LIN {X 0,Y 573.798,Z 251.946,A -85,B 0,C 180,E1 -2291.656,E2 -2291.656} C_VEL
LIN {X 0,Y 573.261,Z 248.706,A -85,B 0,C 180,E1 -2293.069,E2 -2293.069} C_VEL
LIN {X 0,Y 573.229,Z 248.708,A -85,B 0,C 180,E1 -2295.666,E2 -2295.666} C_VEL
LIN {X 0,Y 573.233,Z 248.709,A -85,B 0,C 180,E1 -2298.543,E2 -2298.543} C_VEL
LIN {X 0,Y 573.247,Z 248.707,A -85,B 0,C 180,E1 -2301.298,E2 -2301.298} C_VEL
LIN {X 0,Y 573.218,Z 248.709,A -85,B 0,C 180,E1 -2304.018,E2 -2304.018} C_VEL
LIN {X 0,Y 573.244,Z 248.707,A -85,B 0,C 180,E1 -2306.516,E2 -2306.516} C_VEL
LIN {X 0,Y 573.235,Z 248.708,A -85,B 0,C 180,E1 -2309.118,E2 -2309.118} C_VEL
LIN {X 0,Y 573.255,Z 248.707,A -85,B 0,C 180,E1 -2311.971,E2 -2311.971} C_VEL
LIN {X 0,Y 573.255,Z 248.705,A -85,B 0,C 180,E1 -2314.589,E2 -2314.589} C_VEL
LIN {X 0,Y 573.239,Z 248.706,A -85,B 0,C 180,E1 -2317.662,E2 -2317.662} C_VEL
LIN {X 0,Y 573.285,Z 248.701,A -85,B 0,C 180,E1 -2320.728,E2 -2320.728} C_VEL
LIN {X 0,Y 573.254,Z 248.706,A -85,B 0,C 180,E1 -2323.621,E2 -2323.621} C_VEL
LIN {X 0,Y 573.271,Z 248.703,A -85,B 0,C 180,E1 -2325.806,E2 -2325.806} C_VEL
LIN {X 0,Y 573.268,Z 248.705,A -85,B 0,C 180,E1 -2328.745,E2 -2328.745} C_VEL
LIN {X 0,Y 573.287,Z 248.701,A -85,B 0,C 180,E1 -2331.54,E2 -2331.54} C_VEL
LIN {X 0,Y 573.293,Z 248.7,A -85,B 0,C 180,E1 -2334.371,E2 -2334.371} C_VEL
LIN {X 0,Y 573.314,Z 248.698,A -85,B 0,C 180,E1 -2337.892,E2 -2337.892} C_VEL
LIN {X 0,Y 573.338,Z 248.694,A -85,B 0,C 180,E1 -2340.702,E2 -2340.702} C_VEL
LIN {X 0,Y 573.235,Z 248.708,A -85,B 0,C 180,E1 -2343.514,E2 -2343.514} C_VEL
LIN {X 0,Y 573.29,Z 248.701,A -85,B 0,C 180,E1 -2345.627,E2 -2345.627} C_VEL
LIN {X 0,Y 573.287,Z 248.703,A -85,B 0,C 180,E1 -2348.459,E2 -2348.459} C_VEL
LIN {X 0,Y 573.275,Z 248.702,A -85,B 0,C 180,E1 -2351.311,E2 -2351.311} C_VEL
LIN {X 0,Y 573.284,Z 248.701,A -85,B 0,C 180,E1 -2354.423,E2 -2354.423} C_VEL
LIN {X 0,Y 573.261,Z 248.705,A -85,B 0,C 180,E1 -2357.11,E2 -2357.11} C_VEL
LIN {X 0,Y 573.242,Z 248.709,A -85,B 0,C 180,E1 -2360.076,E2 -2360.076} C_VEL
LIN {X 0,Y 573.237,Z 248.708,A -85,B 0,C 180,E1 -2362.337,E2 -2362.337} C_VEL
LIN {X 0,Y 573.25,Z 248.704,A -85,B 0,C 180,E1 -2364.387,E2 -2364.387} C_VEL
LIN {X 0,Y 572.623,Z 248.784,A -85,B 0,C 180,E1 -2364.973,E2 -2364.973} C_VEL
LIN {X 0,Y 569.781,Z 249.141,A -85,B 0,C 180,E1 -2365.924,E2 -2365.924} C_VEL
LIN {X 0,Y 567.351,Z 249.444,A -85,B 0,C 180,E1 -2366.69,E2 -2366.69} C_VEL
LIN {X 0,Y 566.3,Z 249.573,A -85,B 0,C 180,E1 -2367.281,E2 -2367.281} C_VEL
LIN {X 0,Y 566.212,Z 249.582,A -85,B 0,C 180,E1 -2367.481,E2 -2367.481} C_VEL
LIN {X 0,Y 566.201,Z 249.584,A -85,B 0,C 180,E1 -2369.768,E2 -2369.768} C_VEL
LIN {X 0,Y 566.205,Z 249.584,A -85,B 0,C 180,E1 -2372.429,E2 -2372.429} C_VEL
LIN {X 0,Y 566.212,Z 249.582,A -85,B 0,C 180,E1 -2374.993,E2 -2374.993} C_VEL
LIN {X 0,Y 566.194,Z 249.584,A -85,B 0,C 180,E1 -2377.46,E2 -2377.46} C_VEL
LIN {X 0,Y 566.223,Z 249.581,A -85,B 0,C 180,E1 -2380.196,E2 -2380.196} C_VEL
LIN {X 0,Y 566.201,Z 249.585,A -85,B 0,C 180,E1 -2383.053,E2 -2383.053} C_VEL
LIN {X 0,Y 566.198,Z 249.585,A -85,B 0,C 180,E1 -2386.047,E2 -2386.047} C_VEL
LIN {X 0,Y 566.207,Z 249.582,A -85,B 0,C 180,E1 -2388.863,E2 -2388.863} C_VEL
LIN {X 0,Y 566.184,Z 249.587,A -85,B 0,C 180,E1 -2391.636,E2 -2391.636} C_VEL
LIN {X 0,Y 566.205,Z 249.584,A -85,B 0,C 180,E1 -2394.311,E2 -2394.311} C_VEL
LIN {X 0,Y 566.222,Z 249.581,A -85,B 0,C 180,E1 -2396.898,E2 -2396.898} C_VEL
LIN {X 0,Y 566.188,Z 249.585,A -85,B 0,C 180,E1 -2399.407,E2 -2399.407} C_VEL
LIN {X 0,Y 566.22,Z 249.584,A -85,B 0,C 180,E1 -2401.857,E2 -2401.857} C_VEL
LIN {X 0,Y 566.217,Z 249.581,A -85,B 0,C 180,E1 -2404.251,E2 -2404.251} C_VEL
LIN {X 0,Y 566.184,Z 249.585,A -85,B 0,C 180,E1 -2406.712,E2 -2406.712} C_VEL
LIN {X 0,Y 566.211,Z 249.582,A -85,B 0,C 180,E1 -2409.662,E2 -2409.662} C_VEL
LIN {X 0,Y 566.195,Z 249.584,A -85,B 0,C 180,E1 -2412.668,E2 -2412.668} C_VEL
LIN {X 0,Y 566.224,Z 249.582,A -85,B 0,C 180,E1 -2415.626,E2 -2415.626} C_VEL
LIN {X 0,Y 566.265,Z 249.577,A -85,B 0,C 180,E1 -2418.653,E2 -2418.653} C_VEL
LIN {X 0,Y 566.241,Z 249.579,A -85,B 0,C 180,E1 -2421.434,E2 -2421.434} C_VEL
LIN {X 0,Y 566.254,Z 249.576,A -85,B 0,C 180,E1 -2424.301,E2 -2424.301} C_VEL
LIN {X 0,Y 566.012,Z 249.791,A -85,B 0,C 180,E1 -2426.44,E2 -2426.44} C_VEL
LIN {X 0,Y 566.132,Z 252.646,A -85,B 0,C 180,E1 -2429.288,E2 -2429.288} C_VEL
LIN {X 0,Y 566.053,Z 254.767,A -85,B 0,C 180,E1 -2431.422,E2 -2431.422} C_VEL
LIN {X 0,Y 565.952,Z 257.617,A -85,B 0,C 180,E1 -2434.272,E2 -2434.272} C_VEL
LIN {X 0,Y 565.964,Z 260.459,A -85,B 0,C 180,E1 -2437.133,E2 -2437.133} C_VEL
LIN {X 0,Y 565.884,Z 263.341,A -85,B 0,C 180,E1 -2440.013,E2 -2440.013} C_VEL
LIN {X 0,Y 565.869,Z 265.835,A -85,B 0,C 180,E1 -2442.188,E2 -2442.188} C_VEL
LIN {X 0,Y 565.846,Z 269.385,A -85,B 0,C 180,E1 -2445.234,E2 -2445.234} C_VEL
LIN {X 0,Y 567.922,Z 278.23,A -85,B 0,C 180,E1 -2445.452,E2 -2445.452} C_VEL
LIN {X 0,Y 567.738,Z 293.829,A -85,B 0,C 180,E1 -2445.826,E2 -2445.826} C_VEL
LIN {X 0,Y 567.531,Z 308.287,A -85,B 0,C 180,E1 -2446.316,E2 -2446.316} C_VEL
LIN {X 0,Y 567.321,Z 322.051,A -85,B 0,C 180,E1 -2446.924,E2 -2446.924} C_VEL
LIN {X 0,Y 567.111,Z 335.614,A -85,B 0,C 180,E1 -2447.674,E2 -2447.674} C_VEL
LIN {X 0,Y 566.885,Z 349.436,A -85,B 0,C 180,E1 -2448.616,E2 -2448.616} C_VEL
LIN {X 0,Y 566.624,Z 362.05,A -85,B 0,C 180,E1 -2449.659,E2 -2449.659} C_VEL
LIN {X 0,Y 566.445,Z 372.696,A -85,B 0,C 180,E1 -2450.707,E2 -2450.707} C_VEL
LIN {X 0,Y 566.258,Z 382.584,A -85,B 0,C 180,E1 -2451.859,E2 -2451.859} C_VEL
LIN {X 0,Y 566.15,Z 391.619,A -85,B 0,C 180,E1 -2453.115,E2 -2453.115} C_VEL
LIN {X 0,Y 566.024,Z 400.309,A -85,B 0,C 180,E1 -2454.579,E2 -2454.579} C_VEL
LIN {X 0,Y 565.983,Z 406.016,A -85,B 0,C 180,E1 -2455.76,E2 -2455.76} C_VEL
LIN {X 0,Y 565.926,Z 410.812,A -85,B 0,C 180,E1 -2456.953,E2 -2456.953} C_VEL
LIN {X 0,Y 565.893,Z 415.77,A -85,B 0,C 180,E1 -2458.564,E2 -2458.564} C_VEL
LIN {X 0,Y 565.857,Z 418.497,A -85,B 0,C 180,E1 -2459.788,E2 -2459.788} C_VEL
LIN {X 0,Y 565.854,Z 420.317,A -85,B 0,C 180,E1 -2461.022,E2 -2461.022} C_VEL
LIN {X 0,Y 565.833,Z 421.357,A -85,B 0,C 180,E1 -2462.373,E2 -2462.373} C_VEL
LIN {X 0,Y 565.854,Z 421.235,A -85,B 0,C 180,E1 -2463.98,E2 -2463.98} C_VEL
LIN {X 0,Y 565.843,Z 420.456,A -85,B 0,C 180,E1 -2464.943,E2 -2464.943} C_VEL
LIN {X 0,Y 565.855,Z 417.91,A -85,B 0,C 180,E1 -2466.595,E2 -2466.595} C_VEL
LIN {X 0,Y 565.9,Z 414.68,A -85,B 0,C 180,E1 -2467.933,E2 -2467.933} C_VEL
LIN {X 0,Y 565.934,Z 410.254,A -85,B 0,C 180,E1 -2469.296,E2 -2469.296} C_VEL
LIN {X 0,Y 565.965,Z 404.088,A -85,B 0,C 180,E1 -2470.759,E2 -2470.759} C_VEL
LIN {X 0,Y 566.033,Z 397.007,A -85,B 0,C 180,E1 -2472.103,E2 -2472.103} C_VEL
LIN {X 0,Y 566.146,Z 389.512,A -85,B 0,C 180,E1 -2473.285,E2 -2473.285} C_VEL
LIN {X 0,Y 566.314,Z 380.208,A -85,B 0,C 180,E1 -2474.52,E2 -2474.52} C_VEL
LIN {X 0,Y 566.505,Z 369.066,A -85,B 0,C 180,E1 -2475.756,E2 -2475.756} C_VEL
LIN {X 0,Y 566.73,Z 358.35,A -85,B 0,C 180,E1 -2476.754,E2 -2476.754} C_VEL
LIN {X 0,Y 566.928,Z 345.77,A -85,B 0,C 180,E1 -2477.74,E2 -2477.74} C_VEL
LIN {X 0,Y 567.174,Z 332.538,A -85,B 0,C 180,E1 -2478.596,E2 -2478.596} C_VEL
LIN {X 0,Y 567.408,Z 318.734,A -85,B 0,C 180,E1 -2479.323,E2 -2479.323} C_VEL
LIN {X 0,Y 567.632,Z 304.228,A -85,B 0,C 180,E1 -2479.924,E2 -2479.924} C_VEL
LIN {X 0,Y 567.847,Z 289.312,A -85,B 0,C 180,E1 -2480.387,E2 -2480.387} C_VEL
LIN {X 0,Y 567.764,Z 277.487,A -85,B 0,C 180,E1 -2480.658,E2 -2480.658} C_VEL
LIN {X 0,Y 565.864,Z 269.366,A -85,B 0,C 180,E1 -2480.872,E2 -2480.872} C_VEL
LIN {X 0,Y 565.876,Z 265.917,A -85,B 0,C 180,E1 -2483.83,E2 -2483.83} C_VEL
LIN {X 0,Y 565.881,Z 262.494,A -85,B 0,C 180,E1 -2486.877,E2 -2486.877} C_VEL
LIN {X 0,Y 565.941,Z 260.154,A -85,B 0,C 180,E1 -2489.394,E2 -2489.394} C_VEL
LIN {X 0,Y 565.985,Z 257.918,A -85,B 0,C 180,E1 -2491.846,E2 -2491.846} C_VEL
LIN {X 0,Y 566.067,Z 254.853,A -85,B 0,C 180,E1 -2495.032,E2 -2495.032} C_VEL
LIN {X 0,Y 566.028,Z 252.512,A -85,B 0,C 180,E1 -2497.363,E2 -2497.363} C_VEL
LIN {X 0,Y 566.053,Z 250.266,A -85,B 0,C 180,E1 -2499.658,E2 -2499.658} C_VEL
LIN {X 0,Y 566.089,Z 249.601,A -85,B 0,C 180,E1 -2500.653,E2 -2500.653} C_VEL
LIN {X 0,Y 566.215,Z 249.585,A -85,B 0,C 180,E1 -2503.413,E2 -2503.413} C_VEL
LIN {X 0,Y 566.194,Z 249.585,A -85,B 0,C 180,E1 -2506.36,E2 -2506.36} C_VEL
LIN {X 0,Y 566.228,Z 249.582,A -85,B 0,C 180,E1 -2508.676,E2 -2508.676} C_VEL
LIN {X 0,Y 566.231,Z 249.58,A -85,B 0,C 180,E1 -2511.435,E2 -2511.435} C_VEL
LIN {X 0,Y 566.257,Z 249.577,A -85,B 0,C 180,E1 -2514.303,E2 -2514.303} C_VEL
LIN {X 0,Y 566.28,Z 249.573,A -85,B 0,C 180,E1 -2517.867,E2 -2517.867} C_VEL
LIN {X 0,Y 566.3,Z 249.571,A -85,B 0,C 180,E1 -2520.712,E2 -2520.712} C_VEL
LIN {X 0,Y 566.273,Z 249.575,A -85,B 0,C 180,E1 -2522.846,E2 -2522.846} C_VEL
LIN {X 0,Y 566.258,Z 249.578,A -85,B 0,C 180,E1 -2525.699,E2 -2525.699} C_VEL
LIN {X 0,Y 566.232,Z 249.58,A -85,B 0,C 180,E1 -2528.566,E2 -2528.566} C_VEL
LIN {X 0,Y 566.239,Z 249.578,A -85,B 0,C 180,E1 -2531.455,E2 -2531.455} C_VEL
LIN {X 0,Y 566.232,Z 249.579,A -85,B 0,C 180,E1 -2534.508,E2 -2534.508} C_VEL
LIN {X 0,Y 566.197,Z 249.586,A -85,B 0,C 180,E1 -2537.332,E2 -2537.332} C_VEL
LIN {X 0,Y 566.217,Z 249.583,A -85,B 0,C 180,E1 -2540.338,E2 -2540.338} C_VEL
LIN {X 0,Y 566.187,Z 249.586,A -85,B 0,C 180,E1 -2543.404,E2 -2543.404} C_VEL
LIN {X 0,Y 566.225,Z 249.583,A -85,B 0,C 180,E1 -2545.749,E2 -2545.749} C_VEL
LIN {X 0,Y 566.2,Z 249.584,A -85,B 0,C 180,E1 -2548.203,E2 -2548.203} C_VEL
LIN {X 0,Y 566.189,Z 249.588,A -85,B 0,C 180,E1 -2551.077,E2 -2551.077} C_VEL
LIN {X 0,Y 566.21,Z 249.584,A -85,B 0,C 180,E1 -2553.735,E2 -2553.735} C_VEL
LIN {X 0,Y 566.198,Z 249.586,A -85,B 0,C 180,E1 -2556.57,E2 -2556.57} C_VEL
LIN {X 0,Y 566.22,Z 249.584,A -85,B 0,C 180,E1 -2559.274,E2 -2559.274} C_VEL
LIN {X 0,Y 566.188,Z 249.586,A -85,B 0,C 180,E1 -2562.09,E2 -2562.09} C_VEL
LIN {X 0,Y 566.172,Z 249.588,A -85,B 0,C 180,E1 -2565.036,E2 -2565.036} C_VEL
LIN {X 0,Y 566.255,Z 249.786,A -85,B 0,C 180,E1 -2566.83,E2 -2566.83} C_VEL
LIN {X 0,Y 566.928,Z 254.966,A -85,B 0,C 180,E1 -2568.928,E2 -2568.928} C_VEL
LIN {X 0,Y 566.868,Z 262.764,A -85,B 0,C 180,E1 -2571.692,E2 -2571.692} C_VEL
LIN {X 0,Y 566.755,Z 270.211,A -85,B 0,C 180,E1 -2574.352,E2 -2574.352} C_VEL
LIN {X 0,Y 566.609,Z 277.638,A -85,B 0,C 180,E1 -2576.924,E2 -2576.924} C_VEL
LIN {X 0,Y 566.513,Z 286.302,A -85,B 0,C 180,E1 -2579.84,E2 -2579.84} C_VEL
LIN {X 0,Y 566.398,Z 294.967,A -85,B 0,C 180,E1 -2582.671,E2 -2582.671} C_VEL
LIN {X 0,Y 566.297,Z 303.632,A -85,B 0,C 180,E1 -2585.434,E2 -2585.434} C_VEL
LIN {X 0,Y 566.232,Z 312.296,A -85,B 0,C 180,E1 -2588.14,E2 -2588.14} C_VEL
LIN {X 0,Y 566.146,Z 320.449,A -85,B 0,C 180,E1 -2590.639,E2 -2590.639} C_VEL
LIN {X 0,Y 566.121,Z 325.422,A -85,B 0,C 180,E1 -2592.146,E2 -2592.146} C_VEL
LIN {X 0,Y 567.997,Z 334.459,A -85,B 0,C 180,E1 -2592.341,E2 -2592.341} C_VEL
LIN {X 0,Y 567.864,Z 349.029,A -85,B 0,C 180,E1 -2592.652,E2 -2592.652} C_VEL
LIN {X 0,Y 567.703,Z 363.222,A -85,B 0,C 180,E1 -2593.087,E2 -2593.087} C_VEL
LIN {X 0,Y 567.453,Z 376.838,A -85,B 0,C 180,E1 -2593.635,E2 -2593.635} C_VEL
LIN {X 0,Y 567.219,Z 391.115,A -85,B 0,C 180,E1 -2594.367,E2 -2594.367} C_VEL
LIN {X 0,Y 566.95,Z 404.54,A -85,B 0,C 180,E1 -2595.217,E2 -2595.217} C_VEL
LIN {X 0,Y 566.756,Z 417.173,A -85,B 0,C 180,E1 -2596.19,E2 -2596.19} C_VEL
LIN {X 0,Y 566.545,Z 428.978,A -85,B 0,C 180,E1 -2597.28,E2 -2597.28} C_VEL
LIN {X 0,Y 566.343,Z 438.905,A -85,B 0,C 180,E1 -2598.367,E2 -2598.367} C_VEL
LIN {X 0,Y 566.204,Z 448.622,A -85,B 0,C 180,E1 -2599.632,E2 -2599.632} C_VEL
LIN {X 0,Y 566.079,Z 456.723,A -85,B 0,C 180,E1 -2600.893,E2 -2600.893} C_VEL
LIN {X 0,Y 566.014,Z 463.428,A -85,B 0,C 180,E1 -2602.15,E2 -2602.15} C_VEL
LIN {X 0,Y 565.943,Z 469.609,A -85,B 0,C 180,E1 -2603.584,E2 -2603.584} C_VEL
LIN {X 0,Y 565.867,Z 474.386,A -85,B 0,C 180,E1 -2605.013,E2 -2605.013} C_VEL
LIN {X 0,Y 565.91,Z 477.889,A -85,B 0,C 180,E1 -2606.44,E2 -2606.44} C_VEL
LIN {X 0,Y 565.839,Z 480.194,A -85,B 0,C 180,E1 -2607.865,E2 -2607.865} C_VEL
LIN {X 0,Y 565.837,Z 481.35,A -85,B 0,C 180,E1 -2609.289,E2 -2609.289} C_VEL
LIN {X 0,Y 565.837,Z 481.349,A -85,B 0,C 180,E1 -2610.712,E2 -2610.712} C_VEL
LIN {X 0,Y 565.839,Z 480.192,A -85,B 0,C 180,E1 -2612.136,E2 -2612.136} C_VEL
LIN {X 0,Y 565.91,Z 477.885,A -85,B 0,C 180,E1 -2613.561,E2 -2613.561} C_VEL
LIN {X 0,Y 565.867,Z 474.383,A -85,B 0,C 180,E1 -2614.988,E2 -2614.988} C_VEL
LIN {X 0,Y 565.959,Z 470.923,A -85,B 0,C 180,E1 -2616.059,E2 -2616.059} C_VEL
LIN {X 0,Y 565.998,Z 465.085,A -85,B 0,C 180,E1 -2617.492,E2 -2617.492} C_VEL
LIN {X 0,Y 566.057,Z 457.727,A -85,B 0,C 180,E1 -2618.929,E2 -2618.929} C_VEL
LIN {X 0,Y 566.209,Z 449.853,A -85,B 0,C 180,E1 -2620.188,E2 -2620.188} C_VEL
LIN {X 0,Y 566.31,Z 440.386,A -85,B 0,C 180,E1 -2621.453,E2 -2621.453} C_VEL
LIN {X 0,Y 566.492,Z 430.744,A -85,B 0,C 180,E1 -2622.54,E2 -2622.54} C_VEL
LIN {X 0,Y 566.671,Z 419.283,A -85,B 0,C 180,E1 -2623.63,E2 -2623.63} C_VEL
LIN {X 0,Y 566.929,Z 406.663,A -85,B 0,C 180,E1 -2624.631,E2 -2624.631} C_VEL
LIN {X 0,Y 567.147,Z 394.229,A -85,B 0,C 180,E1 -2625.452,E2 -2625.452} C_VEL
LIN {X 0,Y 567.382,Z 380.751,A -85,B 0,C 180,E1 -2626.183,E2 -2626.183} C_VEL
LIN {X 0,Y 567.634,Z 367.038,A -85,B 0,C 180,E1 -2626.777,E2 -2626.777} C_VEL
LIN {X 0,Y 567.84,Z 351.699,A -85,B 0,C 180,E1 -2627.28,E2 -2627.28} C_VEL
LIN {X 0,Y 567.962,Z 336.542,A -85,B 0,C 180,E1 -2627.626,E2 -2627.626} C_VEL
LIN {X 0,Y 567.707,Z 332.422,A -85,B 0,C 180,E1 -2627.7,E2 -2627.7} C_VEL
LIN {X 0,Y 566.119,Z 325.381,A -85,B 0,C 180,E1 -2627.867,E2 -2627.867} C_VEL
LIN {X 0,Y 566.177,Z 316.006,A -85,B 0,C 180,E1 -2630.719,E2 -2630.719} C_VEL
LIN {X 0,Y 566.31,Z 306.104,A -85,B 0,C 180,E1 -2633.787,E2 -2633.787} C_VEL
LIN {X 0,Y 566.381,Z 296.939,A -85,B 0,C 180,E1 -2636.694,E2 -2636.694} C_VEL
LIN {X 0,Y 566.492,Z 288.814,A -85,B 0,C 180,E1 -2639.331,E2 -2639.331} C_VEL
LIN {X 0,Y 566.566,Z 280.11,A -85,B 0,C 180,E1 -2642.236,E2 -2642.236} C_VEL
LIN {X 0,Y 566.683,Z 271.893,A -85,B 0,C 180,E1 -2645.062,E2 -2645.062} C_VEL
LIN {X 0,Y 566.89,Z 263.99,A -85,B 0,C 180,E1 -2647.856,E2 -2647.856} C_VEL
LIN {X 0,Y 566.923,Z 257.616,A -85,B 0,C 180,E1 -2650.138,E2 -2650.138} C_VEL
LIN {X 0,Y 566.759,Z 252.805,A -85,B 0,C 180,E1 -2651.925,E2 -2651.925} C_VEL
LIN {X 0,Y 566.225,Z 249.583,A -85,B 0,C 180,E1 -2653.296,E2 -2653.296} C_VEL
LIN {X 0,Y 566.199,Z 249.584,A -85,B 0,C 180,E1 -2656.049,E2 -2656.049} C_VEL
LIN {X 0,Y 566.208,Z 249.584,A -85,B 0,C 180,E1 -2659.215,E2 -2659.215} C_VEL
LIN {X 0,Y 566.19,Z 249.586,A -85,B 0,C 180,E1 -2661.637,E2 -2661.637} C_VEL
LIN {X 0,Y 566.168,Z 249.588,A -85,B 0,C 180,E1 -2664.308,E2 -2664.308} C_VEL
LIN {X 0,Y 566.209,Z 249.584,A -85,B 0,C 180,E1 -2666.897,E2 -2666.897} C_VEL
LIN {X 0,Y 566.186,Z 249.585,A -85,B 0,C 180,E1 -2669.407,E2 -2669.407} C_VEL
LIN {X 0,Y 566.217,Z 249.583,A -85,B 0,C 180,E1 -2671.857,E2 -2671.857} C_VEL
LIN {X 0,Y 566.215,Z 249.583,A -85,B 0,C 180,E1 -2674.251,E2 -2674.251} C_VEL
LIN {X 0,Y 566.178,Z 249.586,A -85,B 0,C 180,E1 -2676.718,E2 -2676.718} C_VEL
LIN {X 0,Y 566.218,Z 249.581,A -85,B 0,C 180,E1 -2679.662,E2 -2679.662} C_VEL
LIN {X 0,Y 566.205,Z 249.584,A -85,B 0,C 180,E1 -2682.668,E2 -2682.668} C_VEL
LIN {X 0,Y 566.234,Z 249.581,A -85,B 0,C 180,E1 -2685.626,E2 -2685.626} C_VEL
LIN {X 0,Y 566.24,Z 249.581,A -85,B 0,C 180,E1 -2688.675,E2 -2688.675} C_VEL
LIN {X 0,Y 566.231,Z 249.579,A -85,B 0,C 180,E1 -2691.434,E2 -2691.434} C_VEL
LIN {X 0,Y 566.26,Z 249.576,A -85,B 0,C 180,E1 -2694.301,E2 -2694.301} C_VEL
LIN {X 0,Y 566.285,Z 249.573,A -85,B 0,C 180,E1 -2697.866,E2 -2697.866} C_VEL
LIN {X 0,Y 566.308,Z 249.57,A -85,B 0,C 180,E1 -2700.71,E2 -2700.71} C_VEL
LIN {X 0,Y 566.276,Z 249.574,A -85,B 0,C 180,E1 -2702.845,E2 -2702.845} C_VEL
LIN {X 0,Y 566.259,Z 249.577,A -85,B 0,C 180,E1 -2705.697,E2 -2705.697} C_VEL
LIN {X 0,Y 566.23,Z 249.582,A -85,B 0,C 180,E1 -2708.565,E2 -2708.565} C_VEL
LIN {X 0,Y 566.245,Z 249.578,A -85,B 0,C 180,E1 -2711.453,E2 -2711.453} C_VEL
LIN {X 0,Y 566.237,Z 249.58,A -85,B 0,C 180,E1 -2714.506,E2 -2714.506} C_VEL
LIN {X 0,Y 566.205,Z 249.583,A -85,B 0,C 180,E1 -2717.33,E2 -2717.33} C_VEL
LIN {X 0,Y 566.208,Z 249.583,A -85,B 0,C 180,E1 -2720.336,E2 -2720.336} C_VEL
LIN {X 0,Y 566.19,Z 249.586,A -85,B 0,C 180,E1 -2723.403,E2 -2723.403} C_VEL
LIN {X 0,Y 566.214,Z 249.582,A -85,B 0,C 180,E1 -2725.748,E2 -2725.748} C_VEL
LIN {X 0,Y 566.212,Z 249.582,A -85,B 0,C 180,E1 -2727.481,E2 -2727.481} C_VEL
LIN {X 0,Y 565.535,Z 249.668,A -85,B 0,C 180,E1 -2728.075,E2 -2728.075} C_VEL
LIN {X 0,Y 562.666,Z 250.023,A -85,B 0,C 180,E1 -2729.038,E2 -2729.038} C_VEL
LIN {X 0,Y 560.251,Z 250.325,A -85,B 0,C 180,E1 -2729.814,E2 -2729.814} C_VEL
LIN {X 0,Y 559.221,Z 250.455,A -85,B 0,C 180,E1 -2730.413,E2 -2730.413} C_VEL
LIN {X 0,Y 559.141,Z 250.461,A -85,B 0,C 180,E1 -2730.615,E2 -2730.615} C_VEL
LIN {X 0,Y 559.163,Z 250.461,A -85,B 0,C 180,E1 -2733.573,E2 -2733.573} C_VEL
LIN {X 0,Y 559.167,Z 250.46,A -85,B 0,C 180,E1 -2736.447,E2 -2736.447} C_VEL
LIN {X 0,Y 559.175,Z 250.46,A -85,B 0,C 180,E1 -2738.932,E2 -2738.932} C_VEL
LIN {X 0,Y 559.188,Z 250.458,A -85,B 0,C 180,E1 -2741.766,E2 -2741.766} C_VEL
LIN {X 0,Y 559.135,Z 250.463,A -85,B 0,C 180,E1 -2744.738,E2 -2744.738} C_VEL
LIN {X 0,Y 559.162,Z 250.462,A -85,B 0,C 180,E1 -2747.256,E2 -2747.256} C_VEL
LIN {X 0,Y 559.181,Z 250.459,A -85,B 0,C 180,E1 -2750.134,E2 -2750.134} C_VEL
LIN {X 0,Y 559.14,Z 250.462,A -85,B 0,C 180,E1 -2752.891,E2 -2752.891} C_VEL
LIN {X 0,Y 559.149,Z 250.464,A -85,B 0,C 180,E1 -2755.555,E2 -2755.555} C_VEL
LIN {X 0,Y 559.166,Z 250.46,A -85,B 0,C 180,E1 -2758.137,E2 -2758.137} C_VEL
LIN {X 0,Y 559.151,Z 250.462,A -85,B 0,C 180,E1 -2760.646,E2 -2760.646} C_VEL
LIN {X 0,Y 559.175,Z 250.459,A -85,B 0,C 180,E1 -2763.169,E2 -2763.169} C_VEL
LIN {X 0,Y 559.149,Z 250.462,A -85,B 0,C 180,E1 -2765.494,E2 -2765.494} C_VEL
LIN {X 0,Y 559.168,Z 250.459,A -85,B 0,C 180,E1 -2768.623,E2 -2768.623} C_VEL
LIN {X 0,Y 559.163,Z 250.46,A -85,B 0,C 180,E1 -2770.926,E2 -2770.926} C_VEL
LIN {X 0,Y 559.162,Z 250.46,A -85,B 0,C 180,E1 -2773.947,E2 -2773.947} C_VEL
LIN {X 0,Y 559.166,Z 250.46,A -85,B 0,C 180,E1 -2776.183,E2 -2776.183} C_VEL
LIN {X 0,Y 559.202,Z 250.455,A -85,B 0,C 180,E1 -2779.133,E2 -2779.133} C_VEL
LIN {X 0,Y 559.204,Z 250.454,A -85,B 0,C 180,E1 -2782.053,E2 -2782.053} C_VEL
LIN {X 0,Y 559.214,Z 250.456,A -85,B 0,C 180,E1 -2784.952,E2 -2784.952} C_VEL
LIN {X 0,Y 558.951,Z 250.49,A -85,B 0,C 180,E1 -2786.395,E2 -2786.395} C_VEL
LIN {X 0,Y 559.086,Z 253.286,A -85,B 0,C 180,E1 -2789.279,E2 -2789.279} C_VEL
LIN {X 0,Y 558.997,Z 255.438,A -85,B 0,C 180,E1 -2791.44,E2 -2791.44} C_VEL
LIN {X 0,Y 558.884,Z 258.3,A -85,B 0,C 180,E1 -2794.327,E2 -2794.327} C_VEL
LIN {X 0,Y 558.875,Z 261.141,A -85,B 0,C 180,E1 -2797.224,E2 -2797.224} C_VEL
LIN {X 0,Y 558.817,Z 263.981,A -85,B 0,C 180,E1 -2800.141,E2 -2800.141} C_VEL
LIN {X 0,Y 558.771,Z 266.33,A -85,B 0,C 180,E1 -2802.346,E2 -2802.346} C_VEL
LIN {X 0,Y 558.743,Z 269.365,A -85,B 0,C 180,E1 -2804.982,E2 -2804.982} C_VEL
LIN {X 0,Y 561.182,Z 279.993,A -85,B 0,C 180,E1 -2805.27,E2 -2805.27} C_VEL
LIN {X 0,Y 560.937,Z 295.094,A -85,B 0,C 180,E1 -2805.649,E2 -2805.649} C_VEL
LIN {X 0,Y 560.679,Z 310.405,A -85,B 0,C 180,E1 -2806.194,E2 -2806.194} C_VEL
LIN {X 0,Y 560.416,Z 324.608,A -85,B 0,C 180,E1 -2806.856,E2 -2806.856} C_VEL
LIN {X 0,Y 560.162,Z 338.641,A -85,B 0,C 180,E1 -2807.677,E2 -2807.677} C_VEL
LIN {X 0,Y 559.929,Z 351.182,A -85,B 0,C 180,E1 -2808.571,E2 -2808.571} C_VEL
LIN {X 0,Y 559.608,Z 363.537,A -85,B 0,C 180,E1 -2809.63,E2 -2809.63} C_VEL
LIN {X 0,Y 559.426,Z 374.786,A -85,B 0,C 180,E1 -2810.787,E2 -2810.787} C_VEL
LIN {X 0,Y 559.227,Z 384.6,A -85,B 0,C 180,E1 -2811.987,E2 -2811.987} C_VEL
LIN {X 0,Y 559.101,Z 392.793,A -85,B 0,C 180,E1 -2813.174,E2 -2813.174} C_VEL
LIN {X 0,Y 558.949,Z 400.53,A -85,B 0,C 180,E1 -2814.514,E2 -2814.514} C_VEL
LIN {X 0,Y 558.908,Z 406.206,A -85,B 0,C 180,E1 -2815.71,E2 -2815.71} C_VEL
LIN {X 0,Y 558.836,Z 410.961,A -85,B 0,C 180,E1 -2816.919,E2 -2816.919} C_VEL
LIN {X 0,Y 558.795,Z 415.876,A -85,B 0,C 180,E1 -2818.55,E2 -2818.55} C_VEL
LIN {X 0,Y 558.77,Z 419.252,A -85,B 0,C 180,E1 -2820.205,E2 -2820.205} C_VEL
LIN {X 0,Y 558.75,Z 420.548,A -85,B 0,C 180,E1 -2821.209,E2 -2821.209} C_VEL
LIN {X 0,Y 558.745,Z 421.441,A -85,B 0,C 180,E1 -2822.742,E2 -2822.742} C_VEL
LIN {X 0,Y 558.76,Z 421.301,A -85,B 0,C 180,E1 -2823.89,E2 -2823.89} C_VEL
LIN {X 0,Y 558.74,Z 420.032,A -85,B 0,C 180,E1 -2825.352,E2 -2825.352} C_VEL
LIN {X 0,Y 558.749,Z 418.404,A -85,B 0,C 180,E1 -2826.392,E2 -2826.392} C_VEL
LIN {X 0,Y 558.776,Z 415.746,A -85,B 0,C 180,E1 -2827.594,E2 -2827.594} C_VEL
LIN {X 0,Y 558.851,Z 411.68,A -85,B 0,C 180,E1 -2828.96,E2 -2828.96} C_VEL
LIN {X 0,Y 558.894,Z 406.298,A -85,B 0,C 180,E1 -2830.36,E2 -2830.36} C_VEL
LIN {X 0,Y 558.947,Z 399.385,A -85,B 0,C 180,E1 -2831.789,E2 -2831.789} C_VEL
LIN {X 0,Y 559.102,Z 391.002,A -85,B 0,C 180,E1 -2833.193,E2 -2833.193} C_VEL
LIN {X 0,Y 559.262,Z 381.909,A -85,B 0,C 180,E1 -2834.456,E2 -2834.456} C_VEL
LIN {X 0,Y 559.445,Z 372.126,A -85,B 0,C 180,E1 -2835.602,E2 -2835.602} C_VEL
LIN {X 0,Y 559.712,Z 360.509,A -85,B 0,C 180,E1 -2836.741,E2 -2836.741} C_VEL
LIN {X 0,Y 559.992,Z 347.925,A -85,B 0,C 180,E1 -2837.77,E2 -2837.77} C_VEL
LIN {X 0,Y 560.271,Z 335.564,A -85,B 0,C 180,E1 -2838.611,E2 -2838.611} C_VEL
LIN {X 0,Y 560.537,Z 321.602,A -85,B 0,C 180,E1 -2839.39,E2 -2839.39} C_VEL
LIN {X 0,Y 560.778,Z 306.826,A -85,B 0,C 180,E1 -2840.041,E2 -2840.041} C_VEL
LIN {X 0,Y 561.029,Z 291.201,A -85,B 0,C 180,E1 -2840.555,E2 -2840.555} C_VEL
LIN {X 0,Y 561.046,Z 278.888,A -85,B 0,C 180,E1 -2840.847,E2 -2840.847} C_VEL
LIN {X 0,Y 558.796,Z 269.372,A -85,B 0,C 180,E1 -2841.1,E2 -2841.1} C_VEL
LIN {X 0,Y 558.802,Z 266.305,A -85,B 0,C 180,E1 -2843.765,E2 -2843.765} C_VEL
LIN {X 0,Y 558.831,Z 263.59,A -85,B 0,C 180,E1 -2846.404,E2 -2846.404} C_VEL
LIN {X 0,Y 558.88,Z 261.221,A -85,B 0,C 180,E1 -2848.965,E2 -2848.965} C_VEL
LIN {X 0,Y 558.928,Z 258.728,A -85,B 0,C 180,E1 -2851.663,E2 -2851.663} C_VEL
LIN {X 0,Y 558.982,Z 255.666,A -85,B 0,C 180,E1 -2854.855,E2 -2854.855} C_VEL
LIN {X 0,Y 558.995,Z 253.566,A -85,B 0,C 180,E1 -2857.062,E2 -2857.062} C_VEL
LIN {X 0,Y 558.983,Z 251.27,A -85,B 0,C 180,E1 -2859.389,E2 -2859.389} C_VEL
LIN {X 0,Y 559,Z 250.536,A -85,B 0,C 180,E1 -2860.157,E2 -2860.157} C_VEL
LIN {X 0,Y 559.164,Z 250.461,A -85,B 0,C 180,E1 -2862.787,E2 -2862.787} C_VEL
LIN {X 0,Y 559.189,Z 250.459,A -85,B 0,C 180,E1 -2865.443,E2 -2865.443} C_VEL
LIN {X 0,Y 559.199,Z 250.457,A -85,B 0,C 180,E1 -2868.605,E2 -2868.605} C_VEL
LIN {X 0,Y 559.189,Z 250.457,A -85,B 0,C 180,E1 -2871.327,E2 -2871.327} C_VEL
LIN {X 0,Y 559.227,Z 250.453,A -85,B 0,C 180,E1 -2874.231,E2 -2874.231} C_VEL
LIN {X 0,Y 559.251,Z 250.449,A -85,B 0,C 180,E1 -2877.84,E2 -2877.84} C_VEL
LIN {X 0,Y 559.27,Z 250.447,A -85,B 0,C 180,E1 -2880.721,E2 -2880.721} C_VEL
LIN {X 0,Y 559.239,Z 250.451,A -85,B 0,C 180,E1 -2882.882,E2 -2882.882} C_VEL
LIN {X 0,Y 559.227,Z 250.453,A -85,B 0,C 180,E1 -2885.771,E2 -2885.771} C_VEL
LIN {X 0,Y 559.19,Z 250.458,A -85,B 0,C 180,E1 -2888.675,E2 -2888.675} C_VEL
LIN {X 0,Y 559.202,Z 250.455,A -85,B 0,C 180,E1 -2891.601,E2 -2891.601} C_VEL
LIN {X 0,Y 559.197,Z 250.455,A -85,B 0,C 180,E1 -2894.596,E2 -2894.596} C_VEL
LIN {X 0,Y 559.157,Z 250.461,A -85,B 0,C 180,E1 -2897.558,E2 -2897.558} C_VEL
LIN {X 0,Y 559.184,Z 250.458,A -85,B 0,C 180,E1 -2900.605,E2 -2900.605} C_VEL
LIN {X 0,Y 559.144,Z 250.464,A -85,B 0,C 180,E1 -2903.717,E2 -2903.717} C_VEL
LIN {X 0,Y 559.198,Z 250.456,A -85,B 0,C 180,E1 -2906.097,E2 -2906.097} C_VEL
LIN {X 0,Y 559.161,Z 250.461,A -85,B 0,C 180,E1 -2908.53,E2 -2908.53} C_VEL
LIN {X 0,Y 559.144,Z 250.465,A -85,B 0,C 180,E1 -2911.274,E2 -2911.274} C_VEL
LIN {X 0,Y 559.164,Z 250.463,A -85,B 0,C 180,E1 -2913.95,E2 -2913.95} C_VEL
LIN {X 0,Y 559.139,Z 250.466,A -85,B 0,C 180,E1 -2917.109,E2 -2917.109} C_VEL
LIN {X 0,Y 559.168,Z 250.461,A -85,B 0,C 180,E1 -2919.944,E2 -2919.944} C_VEL
LIN {X 0,Y 559.156,Z 250.464,A -85,B 0,C 180,E1 -2922.744,E2 -2922.744} C_VEL
LIN {X 0,Y 559.154,Z 250.465,A -85,B 0,C 180,E1 -2925.761,E2 -2925.761} C_VEL
LIN {X 0,Y 559.207,Z 250.578,A -85,B 0,C 180,E1 -2926.501,E2 -2926.501} C_VEL
LIN {X 0,Y 559.91,Z 254.9,A -85,B 0,C 180,E1 -2928.299,E2 -2928.299} C_VEL
LIN {X 0,Y 559.972,Z 259.955,A -85,B 0,C 180,E1 -2930.203,E2 -2930.203} C_VEL
LIN {X 0,Y 559.874,Z 267.724,A -85,B 0,C 180,E1 -2932.949,E2 -2932.949} C_VEL
LIN {X 0,Y 559.72,Z 275.162,A -85,B 0,C 180,E1 -2935.596,E2 -2935.596} C_VEL
LIN {X 0,Y 559.572,Z 282.589,A -85,B 0,C 180,E1 -2938.164,E2 -2938.164} C_VEL
LIN {X 0,Y 559.452,Z 291.253,A -85,B 0,C 180,E1 -2941.077,E2 -2941.077} C_VEL
LIN {X 0,Y 559.356,Z 299.918,A -85,B 0,C 180,E1 -2943.912,E2 -2943.912} C_VEL
LIN {X 0,Y 559.246,Z 308.16,A -85,B 0,C 180,E1 -2946.547,E2 -2946.547} C_VEL
LIN {X 0,Y 559.14,Z 317.247,A -85,B 0,C 180,E1 -2949.395,E2 -2949.395} C_VEL
LIN {X 0,Y 559.059,Z 325.424,A -85,B 0,C 180,E1 -2951.913,E2 -2951.913} C_VEL
LIN {X 0,Y 561.238,Z 335.271,A -85,B 0,C 180,E1 -2952.134,E2 -2952.134} C_VEL
LIN {X 0,Y 561.053,Z 350.857,A -85,B 0,C 180,E1 -2952.481,E2 -2952.481} C_VEL
LIN {X 0,Y 560.848,Z 366.218,A -85,B 0,C 180,E1 -2952.983,E2 -2952.983} C_VEL
LIN {X 0,Y 560.538,Z 380.777,A -85,B 0,C 180,E1 -2953.615,E2 -2953.615} C_VEL
LIN {X 0,Y 560.288,Z 394.248,A -85,B 0,C 180,E1 -2954.355,E2 -2954.355} C_VEL
LIN {X 0,Y 559.997,Z 407.551,A -85,B 0,C 180,E1 -2955.249,E2 -2955.249} C_VEL
LIN {X 0,Y 559.702,Z 420.354,A -85,B 0,C 180,E1 -2956.291,E2 -2956.291} C_VEL
LIN {X 0,Y 559.516,Z 430.754,A -85,B 0,C 180,E1 -2957.302,E2 -2957.302} C_VEL
LIN {X 0,Y 559.304,Z 440.395,A -85,B 0,C 180,E1 -2958.402,E2 -2958.402} C_VEL
LIN {X 0,Y 559.168,Z 449.86,A -85,B 0,C 180,E1 -2959.683,E2 -2959.683} C_VEL
LIN {X 0,Y 559.002,Z 457.735,A -85,B 0,C 180,E1 -2960.959,E2 -2960.959} C_VEL
LIN {X 0,Y 558.92,Z 465.091,A -85,B 0,C 180,E1 -2962.414,E2 -2962.414} C_VEL
LIN {X 0,Y 558.86,Z 470.925,A -85,B 0,C 180,E1 -2963.864,E2 -2963.864} C_VEL
LIN {X 0,Y 558.787,Z 474.386,A -85,B 0,C 180,E1 -2964.95,E2 -2964.95} C_VEL
LIN {X 0,Y 558.819,Z 477.889,A -85,B 0,C 180,E1 -2966.395,E2 -2966.395} C_VEL
LIN {X 0,Y 558.745,Z 480.193,A -85,B 0,C 180,E1 -2967.838,E2 -2967.838} C_VEL
LIN {X 0,Y 558.737,Z 481.35,A -85,B 0,C 180,E1 -2969.28,E2 -2969.28} C_VEL
LIN {X 0,Y 558.737,Z 481.349,A -85,B 0,C 180,E1 -2970.721,E2 -2970.721} C_VEL
LIN {X 0,Y 558.745,Z 480.191,A -85,B 0,C 180,E1 -2972.163,E2 -2972.163} C_VEL
LIN {X 0,Y 558.819,Z 477.885,A -85,B 0,C 180,E1 -2973.606,E2 -2973.606} C_VEL
LIN {X 0,Y 558.788,Z 474.383,A -85,B 0,C 180,E1 -2975.051,E2 -2975.051} C_VEL
LIN {X 0,Y 558.844,Z 469.606,A -85,B 0,C 180,E1 -2976.499,E2 -2976.499} C_VEL
LIN {X 0,Y 558.951,Z 463.421,A -85,B 0,C 180,E1 -2977.95,E2 -2977.95} C_VEL
LIN {X 0,Y 559.005,Z 455.647,A -85,B 0,C 180,E1 -2979.407,E2 -2979.407} C_VEL
LIN {X 0,Y 559.217,Z 447.366,A -85,B 0,C 180,E1 -2980.683,E2 -2980.683} C_VEL
LIN {X 0,Y 559.363,Z 437.387,A -85,B 0,C 180,E1 -2981.965,E2 -2981.965} C_VEL
LIN {X 0,Y 559.597,Z 427.186,A -85,B 0,C 180,E1 -2983.066,E2 -2983.066} C_VEL
LIN {X 0,Y 559.826,Z 415.012,A -85,B 0,C 180,E1 -2984.171,E2 -2984.171} C_VEL
LIN {X 0,Y 560.126,Z 402.693,A -85,B 0,C 180,E1 -2985.1,E2 -2985.1} C_VEL
LIN {X 0,Y 560.353,Z 389.513,A -85,B 0,C 180,E1 -2985.924,E2 -2985.924} C_VEL
LIN {X 0,Y 560.658,Z 374.827,A -85,B 0,C 180,E1 -2986.664,E2 -2986.664} C_VEL
LIN {X 0,Y 560.945,Z 359.984,A -85,B 0,C 180,E1 -2987.24,E2 -2987.24} C_VEL
LIN {X 0,Y 561.121,Z 344.417,A -85,B 0,C 180,E1 -2987.682,E2 -2987.682} C_VEL
LIN {X 0,Y 561.076,Z 334.151,A -85,B 0,C 180,E1 -2987.889,E2 -2987.889} C_VEL
LIN {X 0,Y 559.057,Z 325.393,A -85,B 0,C 180,E1 -2988.097,E2 -2988.097} C_VEL
LIN {X 0,Y 559.134,Z 316.006,A -85,B 0,C 180,E1 -2990.992,E2 -2990.992} C_VEL
LIN {X 0,Y 559.276,Z 306.104,A -85,B 0,C 180,E1 -2994.105,E2 -2994.105} C_VEL
LIN {X 0,Y 559.365,Z 298.719,A -85,B 0,C 180,E1 -2996.476,E2 -2996.476} C_VEL
LIN {X 0,Y 559.491,Z 290.012,A -85,B 0,C 180,E1 -2999.334,E2 -2999.334} C_VEL
LIN {X 0,Y 559.597,Z 281.348,A -85,B 0,C 180,E1 -3002.26,E2 -3002.26} C_VEL
LIN {X 0,Y 559.719,Z 273.921,A -85,B 0,C 180,E1 -3004.842,E2 -3004.842} C_VEL
LIN {X 0,Y 559.92,Z 265.741,A -85,B 0,C 180,E1 -3007.743,E2 -3007.743} C_VEL
LIN {X 0,Y 559.98,Z 259.387,A -85,B 0,C 180,E1 -3010.041,E2 -3010.041} C_VEL
LIN {X 0,Y 559.93,Z 254.94,A -85,B 0,C 180,E1 -3011.701,E2 -3011.701} C_VEL
LIN {X 0,Y 559.2,Z 250.458,A -85,B 0,C 180,E1 -3013.619,E2 -3013.619} C_VEL
LIN {X 0,Y 559.149,Z 250.463,A -85,B 0,C 180,E1 -3016.804,E2 -3016.804} C_VEL
LIN {X 0,Y 559.16,Z 250.462,A -85,B 0,C 180,E1 -3019.188,E2 -3019.188} C_VEL
LIN {X 0,Y 559.137,Z 250.463,A -85,B 0,C 180,E1 -3021.982,E2 -3021.982} C_VEL
LIN {X 0,Y 559.137,Z 250.465,A -85,B 0,C 180,E1 -3024.787,E2 -3024.787} C_VEL
LIN {X 0,Y 559.159,Z 250.461,A -85,B 0,C 180,E1 -3027.365,E2 -3027.365} C_VEL
LIN {X 0,Y 559.152,Z 250.462,A -85,B 0,C 180,E1 -3030.143,E2 -3030.143} C_VEL
LIN {X 0,Y 559.176,Z 250.459,A -85,B 0,C 180,E1 -3033.172,E2 -3033.172} C_VEL
LIN {X 0,Y 559.162,Z 250.459,A -85,B 0,C 180,E1 -3035.495,E2 -3035.495} C_VEL
LIN {X 0,Y 559.177,Z 250.459,A -85,B 0,C 180,E1 -3038.624,E2 -3038.624} C_VEL
LIN {X 0,Y 559.174,Z 250.459,A -85,B 0,C 180,E1 -3040.926,E2 -3040.926} C_VEL
LIN {X 0,Y 559.171,Z 250.459,A -85,B 0,C 180,E1 -3043.947,E2 -3043.947} C_VEL
LIN {X 0,Y 559.172,Z 250.459,A -85,B 0,C 180,E1 -3046.183,E2 -3046.183} C_VEL
LIN {X 0,Y 559.211,Z 250.456,A -85,B 0,C 180,E1 -3048.604,E2 -3048.604} C_VEL
LIN {X 0,Y 559.209,Z 250.455,A -85,B 0,C 180,E1 -3052.053,E2 -3052.053} C_VEL
LIN {X 0,Y 559.254,Z 250.451,A -85,B 0,C 180,E1 -3054.953,E2 -3054.953} C_VEL
LIN {X 0,Y 559.256,Z 250.448,A -85,B 0,C 180,E1 -3057.839,E2 -3057.839} C_VEL
LIN {X 0,Y 559.278,Z 250.446,A -85,B 0,C 180,E1 -3060.719,E2 -3060.719} C_VEL
LIN {X 0,Y 559.243,Z 250.45,A -85,B 0,C 180,E1 -3062.881,E2 -3062.881} C_VEL
LIN {X 0,Y 559.228,Z 250.452,A -85,B 0,C 180,E1 -3065.769,E2 -3065.769} C_VEL
LIN {X 0,Y 559.189,Z 250.458,A -85,B 0,C 180,E1 -3068.673,E2 -3068.673} C_VEL
LIN {X 0,Y 559.208,Z 250.455,A -85,B 0,C 180,E1 -3071.599,E2 -3071.599} C_VEL
LIN {X 0,Y 559.202,Z 250.456,A -85,B 0,C 180,E1 -3074.594,E2 -3074.594} C_VEL
LIN {X 0,Y 559.164,Z 250.459,A -85,B 0,C 180,E1 -3077.556,E2 -3077.556} C_VEL
LIN {X 0,Y 559.166,Z 250.46,A -85,B 0,C 180,E1 -3079.837,E2 -3079.837} C_VEL
LIN {X 0,Y 559.142,Z 250.465,A -85,B 0,C 180,E1 -3082.152,E2 -3082.152} C_VEL
LIN {X 0,Y 559.179,Z 250.459,A -85,B 0,C 180,E1 -3085.186,E2 -3085.186} C_VEL
LIN {X 0,Y 559.191,Z 250.457,A -85,B 0,C 180,E1 -3087.71,E2 -3087.71} C_VEL
LIN {X 0,Y 559.141,Z 250.461,A -85,B 0,C 180,E1 -3090.615,E2 -3090.615} C_VEL
LIN {X 0,Y 558.481,Z 250.545,A -85,B 0,C 180,E1 -3091.217,E2 -3091.217} C_VEL
LIN {X 0,Y 555.62,Z 250.902,A -85,B 0,C 180,E1 -3092.193,E2 -3092.193} C_VEL
LIN {X 0,Y 553.208,Z 251.201,A -85,B 0,C 180,E1 -3092.979,E2 -3092.979} C_VEL
LIN {X 0,Y 552.188,Z 251.33,A -85,B 0,C 180,E1 -3093.585,E2 -3093.585} C_VEL
LIN {X 0,Y 552.114,Z 251.336,A -85,B 0,C 180,E1 -3093.791,E2 -3093.791} C_VEL
LIN {X 0,Y 552.109,Z 251.34,A -85,B 0,C 180,E1 -3096.745,E2 -3096.745} C_VEL
LIN {X 0,Y 552.131,Z 251.336,A -85,B 0,C 180,E1 -3099.525,E2 -3099.525} C_VEL
LIN {X 0,Y 552.126,Z 251.336,A -85,B 0,C 180,E1 -3102.424,E2 -3102.424} C_VEL
LIN {X 0,Y 552.095,Z 251.341,A -85,B 0,C 180,E1 -3105.562,E2 -3105.562} C_VEL
LIN {X 0,Y 552.135,Z 251.334,A -85,B 0,C 180,E1 -3108.675,E2 -3108.675} C_VEL
LIN {X 0,Y 552.114,Z 251.34,A -85,B 0,C 180,E1 -3111.41,E2 -3111.41} C_VEL
LIN {X 0,Y 552.106,Z 251.339,A -85,B 0,C 180,E1 -3114.157,E2 -3114.157} C_VEL
LIN {X 0,Y 552.116,Z 251.339,A -85,B 0,C 180,E1 -3116.814,E2 -3116.814} C_VEL
LIN {X 0,Y 552.108,Z 251.339,A -85,B 0,C 180,E1 -3119.391,E2 -3119.391} C_VEL
LIN {X 0,Y 552.12,Z 251.339,A -85,B 0,C 180,E1 -3121.902,E2 -3121.902} C_VEL
LIN {X 0,Y 552.148,Z 251.333,A -85,B 0,C 180,E1 -3124.648,E2 -3124.648} C_VEL
LIN {X 0,Y 552.088,Z 251.342,A -85,B 0,C 180,E1 -3127.548,E2 -3127.548} C_VEL
LIN {X 0,Y 552.14,Z 251.335,A -85,B 0,C 180,E1 -3130.372,E2 -3130.372} C_VEL
LIN {X 0,Y 552.148,Z 251.334,A -85,B 0,C 180,E1 -3132.977,E2 -3132.977} C_VEL
LIN {X 0,Y 552.128,Z 251.336,A -85,B 0,C 180,E1 -3136.004,E2 -3136.004} C_VEL
LIN {X 0,Y 552.169,Z 251.332,A -85,B 0,C 180,E1 -3138.993,E2 -3138.993} C_VEL
LIN {X 0,Y 552.157,Z 251.333,A -85,B 0,C 180,E1 -3141.951,E2 -3141.951} C_VEL
LIN {X 0,Y 552.194,Z 251.33,A -85,B 0,C 180,E1 -3144.888,E2 -3144.888} C_VEL
LIN {X 0,Y 551.912,Z 251.367,A -85,B 0,C 180,E1 -3146.349,E2 -3146.349} C_VEL
LIN {X 0,Y 551.932,Z 252.491,A -85,B 0,C 180,E1 -3147.81,E2 -3147.81} C_VEL
LIN {X 0,Y 552.015,Z 254.667,A -85,B 0,C 180,E1 -3149.999,E2 -3149.999} C_VEL
LIN {X 0,Y 551.785,Z 256.846,A -85,B 0,C 180,E1 -3152.189,E2 -3152.189} C_VEL
LIN {X 0,Y 551.851,Z 259.699,A -85,B 0,C 180,E1 -3155.114,E2 -3155.114} C_VEL
LIN {X 0,Y 551.764,Z 262.582,A -85,B 0,C 180,E1 -3158.054,E2 -3158.054} C_VEL
LIN {X 0,Y 551.748,Z 265.654,A -85,B 0,C 180,E1 -3161.253,E2 -3161.253} C_VEL
LIN {X 0,Y 551.687,Z 269.088,A -85,B 0,C 180,E1 -3164.5,E2 -3164.5} C_VEL
LIN {X 0,Y 551.668,Z 269.386,A -85,B 0,C 180,E1 -3164.761,E2 -3164.761} C_VEL
LIN {X 0,Y 554.387,Z 280.796,A -85,B 0,C 180,E1 -3165.062,E2 -3165.062} C_VEL
LIN {X 0,Y 554.145,Z 296.296,A -85,B 0,C 180,E1 -3165.467,E2 -3165.467} C_VEL
LIN {X 0,Y 553.849,Z 311.367,A -85,B 0,C 180,E1 -3166.02,E2 -3166.02} C_VEL
LIN {X 0,Y 553.542,Z 325.424,A -85,B 0,C 180,E1 -3166.693,E2 -3166.693} C_VEL
LIN {X 0,Y 553.294,Z 338.003,A -85,B 0,C 180,E1 -3167.439,E2 -3167.439} C_VEL
LIN {X 0,Y 553.016,Z 350.503,A -85,B 0,C 180,E1 -3168.332,E2 -3168.332} C_VEL
LIN {X 0,Y 552.687,Z 361.946,A -85,B 0,C 180,E1 -3169.306,E2 -3169.306} C_VEL
LIN {X 0,Y 552.433,Z 373.465,A -85,B 0,C 180,E1 -3170.478,E2 -3170.478} C_VEL
LIN {X 0,Y 552.185,Z 383.594,A -85,B 0,C 180,E1 -3171.707,E2 -3171.707} C_VEL
LIN {X 0,Y 552.053,Z 392.787,A -85,B 0,C 180,E1 -3173.045,E2 -3173.045} C_VEL
LIN {X 0,Y 551.879,Z 400.746,A -85,B 0,C 180,E1 -3174.448,E2 -3174.448} C_VEL
LIN {X 0,Y 551.835,Z 406.395,A -85,B 0,C 180,E1 -3175.658,E2 -3175.658} C_VEL
LIN {X 0,Y 551.74,Z 411.237,A -85,B 0,C 180,E1 -3176.922,E2 -3176.922} C_VEL
LIN {X 0,Y 551.705,Z 415.858,A -85,B 0,C 180,E1 -3178.485,E2 -3178.485} C_VEL
LIN {X 0,Y 551.676,Z 418.952,A -85,B 0,C 180,E1 -3179.974,E2 -3179.974} C_VEL
LIN {X 0,Y 551.635,Z 420.846,A -85,B 0,C 180,E1 -3181.489,E2 -3181.489} C_VEL
LIN {X 0,Y 551.663,Z 421.449,A -85,B 0,C 180,E1 -3182.776,E2 -3182.776} C_VEL
LIN {X 0,Y 551.65,Z 421.175,A -85,B 0,C 180,E1 -3184.099,E2 -3184.099} C_VEL
LIN {X 0,Y 551.662,Z 420.031,A -85,B 0,C 180,E1 -3185.381,E2 -3185.381} C_VEL
LIN {X 0,Y 551.656,Z 417.722,A -85,B 0,C 180,E1 -3186.781,E2 -3186.781} C_VEL
LIN {X 0,Y 551.741,Z 414.274,A -85,B 0,C 180,E1 -3188.199,E2 -3188.199} C_VEL
LIN {X 0,Y 551.788,Z 409.884,A -85,B 0,C 180,E1 -3189.556,E2 -3189.556} C_VEL
LIN {X 0,Y 551.82,Z 404.361,A -85,B 0,C 180,E1 -3190.896,E2 -3190.896} C_VEL
LIN {X 0,Y 551.932,Z 397.958,A -85,B 0,C 180,E1 -3192.163,E2 -3192.163} C_VEL
LIN {X 0,Y 552.079,Z 389.952,A -85,B 0,C 180,E1 -3193.482,E2 -3193.482} C_VEL
LIN {X 0,Y 552.258,Z 380.93,A -85,B 0,C 180,E1 -3194.726,E2 -3194.726} C_VEL
LIN {X 0,Y 552.487,Z 371.016,A -85,B 0,C 180,E1 -3195.879,E2 -3195.879} C_VEL
LIN {X 0,Y 552.773,Z 360.132,A -85,B 0,C 180,E1 -3196.95,E2 -3196.95} C_VEL
LIN {X 0,Y 553.077,Z 347.145,A -85,B 0,C 180,E1 -3198.016,E2 -3198.016} C_VEL
LIN {X 0,Y 553.416,Z 333.818,A -85,B 0,C 180,E1 -3198.916,E2 -3198.916} C_VEL
LIN {X 0,Y 553.712,Z 320.295,A -85,B 0,C 180,E1 -3199.662,E2 -3199.662} C_VEL
LIN {X 0,Y 553.99,Z 306.215,A -85,B 0,C 180,E1 -3200.279,E2 -3200.279} C_VEL
LIN {X 0,Y 554.268,Z 291.005,A -85,B 0,C 180,E1 -3200.781,E2 -3200.781} C_VEL
LIN {X 0,Y 554.269,Z 280.067,A -85,B 0,C 180,E1 -3201.047,E2 -3201.047} C_VEL
LIN {X 0,Y 551.713,Z 269.376,A -85,B 0,C 180,E1 -3201.336,E2 -3201.336} C_VEL
LIN {X 0,Y 551.714,Z 266.398,A -85,B 0,C 180,E1 -3204.13,E2 -3204.13} C_VEL
LIN {X 0,Y 551.746,Z 263.491,A -85,B 0,C 180,E1 -3207.212,E2 -3207.212} C_VEL
LIN {X 0,Y 551.834,Z 260.988,A -85,B 0,C 180,E1 -3209.999,E2 -3209.999} C_VEL
LIN {X 0,Y 551.838,Z 258.457,A -85,B 0,C 180,E1 -3212.712,E2 -3212.712} C_VEL
LIN {X 0,Y 551.925,Z 256.128,A -85,B 0,C 180,E1 -3215.153,E2 -3215.153} C_VEL
LIN {X 0,Y 551.919,Z 253.803,A -85,B 0,C 180,E1 -3217.543,E2 -3217.543} C_VEL
LIN {X 0,Y 551.924,Z 251.556,A -85,B 0,C 180,E1 -3219.892,E2 -3219.892} C_VEL
LIN {X 0,Y 552.047,Z 251.35,A -85,B 0,C 180,E1 -3221.443,E2 -3221.443} C_VEL
LIN {X 0,Y 552.115,Z 251.34,A -85,B 0,C 180,E1 -3223.738,E2 -3223.738} C_VEL
LIN {X 0,Y 552.131,Z 251.336,A -85,B 0,C 180,E1 -3226.005,E2 -3226.005} C_VEL
LIN {X 0,Y 552.157,Z 251.334,A -85,B 0,C 180,E1 -3228.994,E2 -3228.994} C_VEL
LIN {X 0,Y 552.156,Z 251.335,A -85,B 0,C 180,E1 -3231.952,E2 -3231.952} C_VEL
LIN {X 0,Y 552.228,Z 251.325,A -85,B 0,C 180,E1 -3234.89,E2 -3234.89} C_VEL
LIN {X 0,Y 552.222,Z 251.324,A -85,B 0,C 180,E1 -3237.813,E2 -3237.813} C_VEL
LIN {X 0,Y 552.24,Z 251.323,A -85,B 0,C 180,E1 -3240.73,E2 -3240.73} C_VEL
LIN {X 0,Y 552.205,Z 251.327,A -85,B 0,C 180,E1 -3242.919,E2 -3242.919} C_VEL
LIN {X 0,Y 552.197,Z 251.328,A -85,B 0,C 180,E1 -3245.845,E2 -3245.845} C_VEL
LIN {X 0,Y 552.161,Z 251.334,A -85,B 0,C 180,E1 -3248.786,E2 -3248.786} C_VEL
LIN {X 0,Y 552.16,Z 251.333,A -85,B 0,C 180,E1 -3251.751,E2 -3251.751} C_VEL
LIN {X 0,Y 552.134,Z 251.335,A -85,B 0,C 180,E1 -3254.749,E2 -3254.749} C_VEL
LIN {X 0,Y 552.108,Z 251.338,A -85,B 0,C 180,E1 -3257.789,E2 -3257.789} C_VEL
LIN {X 0,Y 552.131,Z 251.336,A -85,B 0,C 180,E1 -3260.102,E2 -3260.102} C_VEL
LIN {X 0,Y 552.095,Z 251.342,A -85,B 0,C 180,E1 -3262.451,E2 -3262.451} C_VEL
LIN {X 0,Y 552.155,Z 251.333,A -85,B 0,C 180,E1 -3265.352,E2 -3265.352} C_VEL
LIN {X 0,Y 552.122,Z 251.338,A -85,B 0,C 180,E1 -3268.098,E2 -3268.098} C_VEL
LIN {X 0,Y 552.1,Z 251.341,A -85,B 0,C 180,E1 -3270.61,E2 -3270.61} C_VEL
LIN {X 0,Y 552.113,Z 251.342,A -85,B 0,C 180,E1 -3273.186,E2 -3273.186} C_VEL
LIN {X 0,Y 552.084,Z 251.344,A -85,B 0,C 180,E1 -3275.844,E2 -3275.844} C_VEL
LIN {X 0,Y 552.124,Z 251.339,A -85,B 0,C 180,E1 -3279.063,E2 -3279.063} C_VEL
LIN {X 0,Y 552.127,Z 251.339,A -85,B 0,C 180,E1 -3281.446,E2 -3281.446} C_VEL
LIN {X 0,Y 552.094,Z 251.342,A -85,B 0,C 180,E1 -3284.532,E2 -3284.532} C_VEL
LIN {X 0,Y 552.16,Z 251.422,A -85,B 0,C 180,E1 -3286.185,E2 -3286.185} C_VEL
LIN {X 0,Y 553.009,Z 257.277,A -85,B 0,C 180,E1 -3288.636,E2 -3288.636} C_VEL
LIN {X 0,Y 552.964,Z 263.086,A -85,B 0,C 180,E1 -3290.832,E2 -3290.832} C_VEL
LIN {X 0,Y 552.88,Z 270.18,A -85,B 0,C 180,E1 -3293.314,E2 -3293.314} C_VEL
LIN {X 0,Y 552.686,Z 277.638,A -85,B 0,C 180,E1 -3295.979,E2 -3295.979} C_VEL
LIN {X 0,Y 552.567,Z 285.064,A -85,B 0,C 180,E1 -3298.57,E2 -3298.57} C_VEL
LIN {X 0,Y 552.452,Z 293.337,A -85,B 0,C 180,E1 -3301.376,E2 -3301.376} C_VEL
LIN {X 0,Y 552.333,Z 302.394,A -85,B 0,C 180,E1 -3304.367,E2 -3304.367} C_VEL
LIN {X 0,Y 552.147,Z 311.058,A -85,B 0,C 180,E1 -3307.157,E2 -3307.157} C_VEL
LIN {X 0,Y 552.073,Z 319.723,A -85,B 0,C 180,E1 -3309.897,E2 -3309.897} C_VEL
LIN {X 0,Y 552.023,Z 325.391,A -85,B 0,C 180,E1 -3311.664,E2 -3311.664} C_VEL
LIN {X 0,Y 554.474,Z 336.051,A -85,B 0,C 180,E1 -3311.921,E2 -3311.921} C_VEL
LIN {X 0,Y 554.261,Z 351.728,A -85,B 0,C 180,E1 -3312.283,E2 -3312.283} C_VEL
LIN {X 0,Y 554.05,Z 366.566,A -85,B 0,C 180,E1 -3312.781,E2 -3312.781} C_VEL
LIN {X 0,Y 553.705,Z 380.779,A -85,B 0,C 180,E1 -3313.407,E2 -3313.407} C_VEL
LIN {X 0,Y 553.412,Z 394.25,A -85,B 0,C 180,E1 -3314.156,E2 -3314.156} C_VEL
LIN {X 0,Y 553.109,Z 407.551,A -85,B 0,C 180,E1 -3315.061,E2 -3315.061} C_VEL
LIN {X 0,Y 552.771,Z 420.354,A -85,B 0,C 180,E1 -3316.115,E2 -3316.115} C_VEL
LIN {X 0,Y 552.529,Z 430.754,A -85,B 0,C 180,E1 -3317.139,E2 -3317.139} C_VEL
LIN {X 0,Y 552.252,Z 441.444,A -85,B 0,C 180,E1 -3318.383,E2 -3318.383} C_VEL
LIN {X 0,Y 552.124,Z 449.861,A -85,B 0,C 180,E1 -3319.55,E2 -3319.55} C_VEL
LIN {X 0,Y 551.958,Z 457.736,A -85,B 0,C 180,E1 -3320.842,E2 -3320.842} C_VEL
LIN {X 0,Y 551.837,Z 465.091,A -85,B 0,C 180,E1 -3322.316,E2 -3322.316} C_VEL
LIN {X 0,Y 551.769,Z 470.574,A -85,B 0,C 180,E1 -3323.681,E2 -3323.681} C_VEL
LIN {X 0,Y 551.713,Z 474.386,A -85,B 0,C 180,E1 -3324.885,E2 -3324.885} C_VEL
LIN {X 0,Y 551.731,Z 477.89,A -85,B 0,C 180,E1 -3326.349,E2 -3326.349} C_VEL
LIN {X 0,Y 551.655,Z 480.193,A -85,B 0,C 180,E1 -3327.81,E2 -3327.81} C_VEL
LIN {X 0,Y 551.637,Z 481.349,A -85,B 0,C 180,E1 -3329.271,E2 -3329.271} C_VEL
LIN {X 0,Y 551.637,Z 481.349,A -85,B 0,C 180,E1 -3330.73,E2 -3330.73} C_VEL
LIN {X 0,Y 551.655,Z 480.191,A -85,B 0,C 180,E1 -3332.191,E2 -3332.191} C_VEL
LIN {X 0,Y 551.731,Z 477.886,A -85,B 0,C 180,E1 -3333.652,E2 -3333.652} C_VEL
LIN {X 0,Y 551.713,Z 474.383,A -85,B 0,C 180,E1 -3335.116,E2 -3335.116} C_VEL
LIN {X 0,Y 551.781,Z 469.606,A -85,B 0,C 180,E1 -3336.583,E2 -3336.583} C_VEL
LIN {X 0,Y 551.877,Z 463.421,A -85,B 0,C 180,E1 -3338.053,E2 -3338.053} C_VEL
LIN {X 0,Y 551.951,Z 455.647,A -85,B 0,C 180,E1 -3339.528,E2 -3339.528} C_VEL
LIN {X 0,Y 552.184,Z 447.366,A -85,B 0,C 180,E1 -3340.821,E2 -3340.821} C_VEL
LIN {X 0,Y 552.354,Z 437.387,A -85,B 0,C 180,E1 -3342.119,E2 -3342.119} C_VEL
LIN {X 0,Y 552.609,Z 427.185,A -85,B 0,C 180,E1 -3343.234,E2 -3343.234} C_VEL
LIN {X 0,Y 552.89,Z 415.013,A -85,B 0,C 180,E1 -3344.352,E2 -3344.352} C_VEL
LIN {X 0,Y 553.226,Z 402.445,A -85,B 0,C 180,E1 -3345.311,E2 -3345.311} C_VEL
LIN {X 0,Y 553.495,Z 389.511,A -85,B 0,C 180,E1 -3346.127,E2 -3346.127} C_VEL
LIN {X 0,Y 553.813,Z 374.825,A -85,B 0,C 180,E1 -3346.876,E2 -3346.876} C_VEL
LIN {X 0,Y 554.147,Z 359.55,A -85,B 0,C 180,E1 -3347.474,E2 -3347.474} C_VEL
LIN {X 0,Y 554.384,Z 343.63,A -85,B 0,C 180,E1 -3347.924,E2 -3347.924} C_VEL
LIN {X 0,Y 554.257,Z 334.933,A -85,B 0,C 180,E1 -3348.104,E2 -3348.104} C_VEL
LIN {X 0,Y 552.019,Z 325.393,A -85,B 0,C 180,E1 -3348.335,E2 -3348.335} C_VEL
LIN {X 0,Y 552.129,Z 316.006,A -85,B 0,C 180,E1 -3351.271,E2 -3351.271} C_VEL
LIN {X 0,Y 552.242,Z 306.104,A -85,B 0,C 180,E1 -3354.432,E2 -3354.432} C_VEL
LIN {X 0,Y 552.361,Z 298.094,A -85,B 0,C 180,E1 -3357.045,E2 -3357.045} C_VEL
LIN {X 0,Y 552.498,Z 290.012,A -85,B 0,C 180,E1 -3359.742,E2 -3359.742} C_VEL
LIN {X 0,Y 552.627,Z 282.585,A -85,B 0,C 180,E1 -3362.286,E2 -3362.286} C_VEL
LIN {X 0,Y 552.75,Z 275.159,A -85,B 0,C 180,E1 -3364.901,E2 -3364.901} C_VEL
LIN {X 0,Y 552.947,Z 267.579,A -85,B 0,C 180,E1 -3367.596,E2 -3367.596} C_VEL
LIN {X 0,Y 553.036,Z 259.932,A -85,B 0,C 180,E1 -3370.4,E2 -3370.4} C_VEL
LIN {X 0,Y 552.959,Z 256.099,A -85,B 0,C 180,E1 -3371.856,E2 -3371.856} C_VEL
LIN {X 0,Y 552.141,Z 251.337,A -85,B 0,C 180,E1 -3373.996,E2 -3373.996} C_VEL
LIN {X 0,Y 552.111,Z 251.34,A -85,B 0,C 180,E1 -3376.576,E2 -3376.576} C_VEL
LIN {X 0,Y 552.113,Z 251.34,A -85,B 0,C 180,E1 -3379.519,E2 -3379.519} C_VEL
LIN {X 0,Y 552.097,Z 251.341,A -85,B 0,C 180,E1 -3382.336,E2 -3382.336} C_VEL
LIN {X 0,Y 552.088,Z 251.342,A -85,B 0,C 180,E1 -3385.051,E2 -3385.051} C_VEL
LIN {X 0,Y 552.12,Z 251.339,A -85,B 0,C 180,E1 -3387.681,E2 -3387.681} C_VEL
LIN {X 0,Y 552.115,Z 251.338,A -85,B 0,C 180,E1 -3390.235,E2 -3390.235} C_VEL
LIN {X 0,Y 552.145,Z 251.337,A -85,B 0,C 180,E1 -3393,E2 -3393} C_VEL
LIN {X 0,Y 552.119,Z 251.339,A -85,B 0,C 180,E1 -3395.161,E2 -3395.161} C_VEL
LIN {X 0,Y 552.132,Z 251.338,A -85,B 0,C 180,E1 -3398.337,E2 -3398.337} C_VEL
LIN {X 0,Y 552.162,Z 251.333,A -85,B 0,C 180,E1 -3400.674,E2 -3400.674} C_VEL
LIN {X 0,Y 552.121,Z 251.337,A -85,B 0,C 180,E1 -3403.737,E2 -3403.737} C_VEL
LIN {X 0,Y 552.138,Z 251.335,A -85,B 0,C 180,E1 -3406.004,E2 -3406.004} C_VEL
LIN {X 0,Y 552.166,Z 251.332,A -85,B 0,C 180,E1 -3408.993,E2 -3408.993} C_VEL
LIN {X 0,Y 552.163,Z 251.334,A -85,B 0,C 180,E1 -3411.951,E2 -3411.951} C_VEL
LIN {X 0,Y 552.229,Z 251.326,A -85,B 0,C 180,E1 -3414.888,E2 -3414.888} C_VEL
LIN {X 0,Y 552.228,Z 251.324,A -85,B 0,C 180,E1 -3417.811,E2 -3417.811} C_VEL
LIN {X 0,Y 552.248,Z 251.322,A -85,B 0,C 180,E1 -3420.728,E2 -3420.728} C_VEL
LIN {X 0,Y 552.209,Z 251.326,A -85,B 0,C 180,E1 -3422.917,E2 -3422.917} C_VEL
LIN {X 0,Y 552.199,Z 251.328,A -85,B 0,C 180,E1 -3425.843,E2 -3425.843} C_VEL
LIN {X 0,Y 552.16,Z 251.333,A -85,B 0,C 180,E1 -3428.785,E2 -3428.785} C_VEL
LIN {X 0,Y 552.165,Z 251.334,A -85,B 0,C 180,E1 -3431.749,E2 -3431.749} C_VEL
LIN {X 0,Y 552.139,Z 251.337,A -85,B 0,C 180,E1 -3434.747,E2 -3434.747} C_VEL
LIN {X 0,Y 552.115,Z 251.339,A -85,B 0,C 180,E1 -3437.787,E2 -3437.787} C_VEL
LIN {X 0,Y 552.127,Z 251.339,A -85,B 0,C 180,E1 -3440.1,E2 -3440.1} C_VEL
LIN {X 0,Y 552.096,Z 251.341,A -85,B 0,C 180,E1 -3442.45,E2 -3442.45} C_VEL
LIN {X 0,Y 552.155,Z 251.334,A -85,B 0,C 180,E1 -3445.349,E2 -3445.349} C_VEL
LIN {X 0,Y 552.125,Z 251.337,A -85,B 0,C 180,E1 -3448.096,E2 -3448.096} C_VEL
LIN {X 0,Y 552.103,Z 251.34,A -85,B 0,C 180,E1 -3450.611,E2 -3450.611} C_VEL
LIN {X 0,Y 552.121,Z 251.336,A -85,B 0,C 180,E1 -3453.184,E2 -3453.184} C_VEL
LIN {X 0,Y 552.114,Z 251.336,A -85,B 0,C 180,E1 -3453.791,E2 -3453.791} C_VEL
LIN {X 0,Y 551.478,Z 251.418,A -85,B 0,C 180,E1 -3454.4,E2 -3454.4} C_VEL
LIN {X 0,Y 548.656,Z 251.773,A -85,B 0,C 180,E1 -3455.388,E2 -3455.388} C_VEL
LIN {X 0,Y 546.235,Z 252.074,A -85,B 0,C 180,E1 -3456.183,E2 -3456.183} C_VEL
LIN {X 0,Y 545.165,Z 252.205,A -85,B 0,C 180,E1 -3456.797,E2 -3456.797} C_VEL
LIN {X 0,Y 545.063,Z 252.217,A -85,B 0,C 180,E1 -3457.005,E2 -3457.005} C_VEL
LIN {X 0,Y 545.071,Z 252.216,A -85,B 0,C 180,E1 -3460.14,E2 -3460.14} C_VEL
LIN {X 0,Y 545.082,Z 252.215,A -85,B 0,C 180,E1 -3463.105,E2 -3463.105} C_VEL
LIN {X 0,Y 545.061,Z 252.218,A -85,B 0,C 180,E1 -3466.223,E2 -3466.223} C_VEL
LIN {X 0,Y 545.096,Z 252.211,A -85,B 0,C 180,E1 -3468.886,E2 -3468.886} C_VEL
LIN {X 0,Y 545.048,Z 252.219,A -85,B 0,C 180,E1 -3471.762,E2 -3471.762} C_VEL
LIN {X 0,Y 545.058,Z 252.218,A -85,B 0,C 180,E1 -3474.533,E2 -3474.533} C_VEL
LIN {X 0,Y 545.075,Z 252.215,A -85,B 0,C 180,E1 -3477.211,E2 -3477.211} C_VEL
LIN {X 0,Y 545.094,Z 252.215,A -85,B 0,C 180,E1 -3479.812,E2 -3479.812} C_VEL
LIN {X 0,Y 545.094,Z 252.213,A -85,B 0,C 180,E1 -3482.824,E2 -3482.824} C_VEL
LIN {X 0,Y 545.044,Z 252.219,A -85,B 0,C 180,E1 -3485.63,E2 -3485.63} C_VEL
LIN {X 0,Y 545.061,Z 252.216,A -85,B 0,C 180,E1 -3488.836,E2 -3488.836} C_VEL
LIN {X 0,Y 545.076,Z 252.216,A -85,B 0,C 180,E1 -3491.195,E2 -3491.195} C_VEL
LIN {X 0,Y 545.068,Z 252.217,A -85,B 0,C 180,E1 -3493.521,E2 -3493.521} C_VEL
LIN {X 0,Y 545.086,Z 252.214,A -85,B 0,C 180,E1 -3495.819,E2 -3495.819} C_VEL
LIN {X 0,Y 545.123,Z 252.21,A -85,B 0,C 180,E1 -3498.849,E2 -3498.849} C_VEL
LIN {X 0,Y 545.127,Z 252.209,A -85,B 0,C 180,E1 -3501.847,E2 -3501.847} C_VEL
LIN {X 0,Y 545.154,Z 252.206,A -85,B 0,C 180,E1 -3504.822,E2 -3504.822} C_VEL
LIN {X 0,Y 544.803,Z 252.442,A -85,B 0,C 180,E1 -3507.042,E2 -3507.042} C_VEL
LIN {X 0,Y 544.998,Z 254.623,A -85,B 0,C 180,E1 -3509.261,E2 -3509.261} C_VEL
LIN {X 0,Y 544.842,Z 256.791,A -85,B 0,C 180,E1 -3511.478,E2 -3511.478} C_VEL
LIN {X 0,Y 544.756,Z 259.69,A -85,B 0,C 180,E1 -3514.439,E2 -3514.439} C_VEL
LIN {X 0,Y 544.747,Z 262.591,A -85,B 0,C 180,E1 -3517.412,E2 -3517.412} C_VEL
LIN {X 0,Y 544.699,Z 265.503,A -85,B 0,C 180,E1 -3520.406,E2 -3520.406} C_VEL
LIN {X 0,Y 544.581,Z 268.416,A -85,B 0,C 180,E1 -3523.432,E2 -3523.432} C_VEL
LIN {X 0,Y 544.619,Z 269.472,A -85,B 0,C 180,E1 -3524.511,E2 -3524.511} C_VEL
LIN {X 0,Y 547.646,Z 282.618,A -85,B 0,C 180,E1 -3524.872,E2 -3524.872} C_VEL
LIN {X 0,Y 547.333,Z 297.777,A -85,B 0,C 180,E1 -3525.288,E2 -3525.288} C_VEL
LIN {X 0,Y 547.014,Z 312.355,A -85,B 0,C 180,E1 -3525.843,E2 -3525.843} C_VEL
LIN {X 0,Y 546.68,Z 326.201,A -85,B 0,C 180,E1 -3526.524,E2 -3526.524} C_VEL
LIN {X 0,Y 546.38,Z 339.718,A -85,B 0,C 180,E1 -3527.352,E2 -3527.352} C_VEL
LIN {X 0,Y 546.069,Z 352.244,A -85,B 0,C 180,E1 -3528.282,E2 -3528.282} C_VEL
LIN {X 0,Y 545.67,Z 364.438,A -85,B 0,C 180,E1 -3529.368,E2 -3529.368} C_VEL
LIN {X 0,Y 545.406,Z 375.558,A -85,B 0,C 180,E1 -3530.556,E2 -3530.556} C_VEL
LIN {X 0,Y 545.141,Z 385.647,A -85,B 0,C 180,E1 -3531.844,E2 -3531.844} C_VEL
LIN {X 0,Y 544.983,Z 394.256,A -85,B 0,C 180,E1 -3533.161,E2 -3533.161} C_VEL
LIN {X 0,Y 544.832,Z 400.956,A -85,B 0,C 180,E1 -3534.379,E2 -3534.379} C_VEL
LIN {X 0,Y 544.762,Z 406.964,A -85,B 0,C 180,E1 -3535.693,E2 -3535.693} C_VEL
LIN {X 0,Y 544.662,Z 412.058,A -85,B 0,C 180,E1 -3537.088,E2 -3537.088} C_VEL
LIN {X 0,Y 544.616,Z 416.423,A -85,B 0,C 180,E1 -3538.66,E2 -3538.66} C_VEL
LIN {X 0,Y 544.581,Z 419.382,A -85,B 0,C 180,E1 -3540.218,E2 -3540.218} C_VEL
LIN {X 0,Y 544.544,Z 421.156,A -85,B 0,C 180,E1 -3541.948,E2 -3541.948} C_VEL
LIN {X 0,Y 544.561,Z 421.493,A -85,B 0,C 180,E1 -3542.981,E2 -3542.981} C_VEL
LIN {X 0,Y 544.554,Z 420.86,A -85,B 0,C 180,E1 -3544.601,E2 -3544.601} C_VEL
LIN {X 0,Y 544.554,Z 419.786,A -85,B 0,C 180,E1 -3545.605,E2 -3545.605} C_VEL
LIN {X 0,Y 544.572,Z 417.665,A -85,B 0,C 180,E1 -3546.859,E2 -3546.859} C_VEL
LIN {X 0,Y 544.652,Z 414.265,A -85,B 0,C 180,E1 -3548.27,E2 -3548.27} C_VEL
LIN {X 0,Y 544.692,Z 409.678,A -85,B 0,C 180,E1 -3549.695,E2 -3549.695} C_VEL
LIN {X 0,Y 544.737,Z 403.706,A -85,B 0,C 180,E1 -3551.145,E2 -3551.145} C_VEL
LIN {X 0,Y 544.882,Z 397.309,A -85,B 0,C 180,E1 -3552.402,E2 -3552.402} C_VEL
LIN {X 0,Y 545.064,Z 388.906,A -85,B 0,C 180,E1 -3553.777,E2 -3553.777} C_VEL
LIN {X 0,Y 545.271,Z 380.226,A -85,B 0,C 180,E1 -3554.967,E2 -3554.967} C_VEL
LIN {X 0,Y 545.541,Z 369.832,A -85,B 0,C 180,E1 -3556.171,E2 -3556.171} C_VEL
LIN {X 0,Y 545.886,Z 358.398,A -85,B 0,C 180,E1 -3557.283,E2 -3557.283} C_VEL
LIN {X 0,Y 546.205,Z 346.333,A -85,B 0,C 180,E1 -3558.268,E2 -3558.268} C_VEL
LIN {X 0,Y 546.566,Z 333.828,A -85,B 0,C 180,E1 -3559.12,E2 -3559.12} C_VEL
LIN {X 0,Y 546.868,Z 320.992,A -85,B 0,C 180,E1 -3559.842,E2 -3559.842} C_VEL
LIN {X 0,Y 547.197,Z 306.092,A -85,B 0,C 180,E1 -3560.505,E2 -3560.505} C_VEL
LIN {X 0,Y 547.529,Z 291.008,A -85,B 0,C 180,E1 -3561.007,E2 -3561.007} C_VEL
LIN {X 0,Y 547.435,Z 281.147,A -85,B 0,C 180,E1 -3561.257,E2 -3561.257} C_VEL
LIN {X 0,Y 544.601,Z 269.499,A -85,B 0,C 180,E1 -3561.58,E2 -3561.58} C_VEL
LIN {X 0,Y 544.656,Z 266.661,A -85,B 0,C 180,E1 -3564.505,E2 -3564.505} C_VEL
LIN {X 0,Y 544.686,Z 264.236,A -85,B 0,C 180,E1 -3567.187,E2 -3567.187} C_VEL
LIN {X 0,Y 544.784,Z 261.909,A -85,B 0,C 180,E1 -3569.806,E2 -3569.806} C_VEL
LIN {X 0,Y 544.776,Z 259.545,A -85,B 0,C 180,E1 -3572.328,E2 -3572.328} C_VEL
LIN {X 0,Y 544.868,Z 256.43,A -85,B 0,C 180,E1 -3575.623,E2 -3575.623} C_VEL
LIN {X 0,Y 544.903,Z 253.96,A -85,B 0,C 180,E1 -3578.221,E2 -3578.221} C_VEL
LIN {X 0,Y 544.851,Z 252.589,A -85,B 0,C 180,E1 -3579.62,E2 -3579.62} C_VEL
LIN {X 0,Y 544.945,Z 252.235,A -85,B 0,C 180,E1 -3580.409,E2 -3580.409} C_VEL
LIN {X 0,Y 545.07,Z 252.217,A -85,B 0,C 180,E1 -3582.75,E2 -3582.75} C_VEL
LIN {X 0,Y 545.09,Z 252.214,A -85,B 0,C 180,E1 -3585.821,E2 -3585.821} C_VEL
LIN {X 0,Y 545.112,Z 252.212,A -85,B 0,C 180,E1 -3588.85,E2 -3588.85} C_VEL
LIN {X 0,Y 545.126,Z 252.211,A -85,B 0,C 180,E1 -3591.848,E2 -3591.848} C_VEL
LIN {X 0,Y 545.203,Z 252.199,A -85,B 0,C 180,E1 -3594.824,E2 -3594.824} C_VEL
LIN {X 0,Y 545.194,Z 252.199,A -85,B 0,C 180,E1 -3597.784,E2 -3597.784} C_VEL
LIN {X 0,Y 545.21,Z 252.198,A -85,B 0,C 180,E1 -3600.739,E2 -3600.739} C_VEL
LIN {X 0,Y 545.171,Z 252.203,A -85,B 0,C 180,E1 -3602.957,E2 -3602.957} C_VEL
LIN {X 0,Y 545.169,Z 252.203,A -85,B 0,C 180,E1 -3605.92,E2 -3605.92} C_VEL
LIN {X 0,Y 545.12,Z 252.211,A -85,B 0,C 180,E1 -3608.901,E2 -3608.901} C_VEL
LIN {X 0,Y 545.132,Z 252.209,A -85,B 0,C 180,E1 -3611.905,E2 -3611.905} C_VEL
LIN {X 0,Y 545.083,Z 252.214,A -85,B 0,C 180,E1 -3614.944,E2 -3614.944} C_VEL
LIN {X 0,Y 545.076,Z 252.215,A -85,B 0,C 180,E1 -3618.026,E2 -3618.026} C_VEL
LIN {X 0,Y 545.096,Z 252.214,A -85,B 0,C 180,E1 -3620.373,E2 -3620.373} C_VEL
LIN {X 0,Y 545.089,Z 252.214,A -85,B 0,C 180,E1 -3623.559,E2 -3623.559} C_VEL
LIN {X 0,Y 545.087,Z 252.214,A -85,B 0,C 180,E1 -3626.001,E2 -3626.001} C_VEL
LIN {X 0,Y 545.087,Z 252.216,A -85,B 0,C 180,E1 -3628.749,E2 -3628.749} C_VEL
LIN {X 0,Y 545.055,Z 252.22,A -85,B 0,C 180,E1 -3631.679,E2 -3631.679} C_VEL
LIN {X 0,Y 545.061,Z 252.22,A -85,B 0,C 180,E1 -3634.565,E2 -3634.565} C_VEL
LIN {X 0,Y 545.035,Z 252.224,A -85,B 0,C 180,E1 -3637.305,E2 -3637.305} C_VEL
LIN {X 0,Y 545.072,Z 252.217,A -85,B 0,C 180,E1 -3640.142,E2 -3640.142} C_VEL
LIN {X 0,Y 545.076,Z 252.217,A -85,B 0,C 180,E1 -3643.107,E2 -3643.107} C_VEL
LIN {X 0,Y 545.108,Z 252.284,A -85,B 0,C 180,E1 -3645.877,E2 -3645.877} C_VEL
LIN {X 0,Y 546.034,Z 257.954,A -85,B 0,C 180,E1 -3648.29,E2 -3648.29} C_VEL
LIN {X 0,Y 546.016,Z 263.655,A -85,B 0,C 180,E1 -3650.56,E2 -3650.56} C_VEL
LIN {X 0,Y 545.886,Z 271.475,A -85,B 0,C 180,E1 -3653.321,E2 -3653.321} C_VEL
LIN {X 0,Y 545.723,Z 278.894,A -85,B 0,C 180,E1 -3655.937,E2 -3655.937} C_VEL
LIN {X 0,Y 545.565,Z 286.451,A -85,B 0,C 180,E1 -3658.605,E2 -3658.605} C_VEL
LIN {X 0,Y 545.436,Z 294.967,A -85,B 0,C 180,E1 -3661.527,E2 -3661.527} C_VEL
LIN {X 0,Y 545.297,Z 303.71,A -85,B 0,C 180,E1 -3664.447,E2 -3664.447} C_VEL
LIN {X 0,Y 545.127,Z 312.296,A -85,B 0,C 180,E1 -3667.247,E2 -3667.247} C_VEL
LIN {X 0,Y 545.025,Z 320.893,A -85,B 0,C 180,E1 -3669.998,E2 -3669.998} C_VEL
LIN {X 0,Y 544.995,Z 325.416,A -85,B 0,C 180,E1 -3671.427,E2 -3671.427} C_VEL
LIN {X 0,Y 547.698,Z 337.725,A -85,B 0,C 180,E1 -3671.725,E2 -3671.725} C_VEL
LIN {X 0,Y 547.486,Z 352.854,A -85,B 0,C 180,E1 -3672.092,E2 -3672.092} C_VEL
LIN {X 0,Y 547.263,Z 366.893,A -85,B 0,C 180,E1 -3672.573,E2 -3672.573} C_VEL
LIN {X 0,Y 546.878,Z 380.78,A -85,B 0,C 180,E1 -3673.193,E2 -3673.193} C_VEL
LIN {X 0,Y 546.546,Z 394.251,A -85,B 0,C 180,E1 -3673.951,E2 -3673.951} C_VEL
LIN {X 0,Y 546.229,Z 406.536,A -85,B 0,C 180,E1 -3674.792,E2 -3674.792} C_VEL
LIN {X 0,Y 545.846,Z 419.295,A -85,B 0,C 180,E1 -3675.84,E2 -3675.84} C_VEL
LIN {X 0,Y 545.567,Z 430.754,A -85,B 0,C 180,E1 -3676.972,E2 -3676.972} C_VEL
LIN {X 0,Y 545.281,Z 440.395,A -85,B 0,C 180,E1 -3678.1,E2 -3678.1} C_VEL
LIN {X 0,Y 545.085,Z 449.861,A -85,B 0,C 180,E1 -3679.413,E2 -3679.413} C_VEL
LIN {X 0,Y 544.899,Z 457.736,A -85,B 0,C 180,E1 -3680.723,E2 -3680.723} C_VEL
LIN {X 0,Y 544.772,Z 465.091,A -85,B 0,C 180,E1 -3682.215,E2 -3682.215} C_VEL
LIN {X 0,Y 544.675,Z 470.92,A -85,B 0,C 180,E1 -3683.702,E2 -3683.702} C_VEL
LIN {X 0,Y 544.642,Z 474.387,A -85,B 0,C 180,E1 -3684.818,E2 -3684.818} C_VEL
LIN {X 0,Y 544.645,Z 477.89,A -85,B 0,C 180,E1 -3686.301,E2 -3686.301} C_VEL
LIN {X 0,Y 544.569,Z 480.193,A -85,B 0,C 180,E1 -3687.782,E2 -3687.782} C_VEL
LIN {X 0,Y 544.537,Z 481.349,A -85,B 0,C 180,E1 -3689.261,E2 -3689.261} C_VEL
LIN {X 0,Y 544.537,Z 481.349,A -85,B 0,C 180,E1 -3690.74,E2 -3690.74} C_VEL
LIN {X 0,Y 544.569,Z 480.19,A -85,B 0,C 180,E1 -3692.219,E2 -3692.219} C_VEL
LIN {X 0,Y 544.645,Z 477.886,A -85,B 0,C 180,E1 -3693.7,E2 -3693.7} C_VEL
LIN {X 0,Y 544.642,Z 474.384,A -85,B 0,C 180,E1 -3695.183,E2 -3695.183} C_VEL
LIN {X 0,Y 544.699,Z 469.606,A -85,B 0,C 180,E1 -3696.669,E2 -3696.669} C_VEL
LIN {X 0,Y 544.819,Z 463.421,A -85,B 0,C 180,E1 -3698.158,E2 -3698.158} C_VEL
LIN {X 0,Y 544.905,Z 455.646,A -85,B 0,C 180,E1 -3699.653,E2 -3699.653} C_VEL
LIN {X 0,Y 545.15,Z 447.366,A -85,B 0,C 180,E1 -3700.962,E2 -3700.962} C_VEL
LIN {X 0,Y 545.359,Z 437.387,A -85,B 0,C 180,E1 -3702.277,E2 -3702.277} C_VEL
LIN {X 0,Y 545.64,Z 427.185,A -85,B 0,C 180,E1 -3703.406,E2 -3703.406} C_VEL
LIN {X 0,Y 545.973,Z 415.013,A -85,B 0,C 180,E1 -3704.538,E2 -3704.538} C_VEL
LIN {X 0,Y 546.355,Z 402.648,A -85,B 0,C 180,E1 -3705.493,E2 -3705.493} C_VEL
LIN {X 0,Y 546.653,Z 389.51,A -85,B 0,C 180,E1 -3706.334,E2 -3706.334} C_VEL
LIN {X 0,Y 547.014,Z 374.824,A -85,B 0,C 180,E1 -3707.092,E2 -3707.092} C_VEL
LIN {X 0,Y 547.363,Z 360.284,A -85,B 0,C 180,E1 -3707.671,E2 -3707.671} C_VEL
LIN {X 0,Y 547.604,Z 344.983,A -85,B 0,C 180,E1 -3708.119,E2 -3708.119} C_VEL
LIN {X 0,Y 547.598,Z 336.468,A -85,B 0,C 180,E1 -3708.305,E2 -3708.305} C_VEL
LIN {X 0,Y 544.966,Z 325.347,A -85,B 0,C 180,E1 -3708.596,E2 -3708.596} C_VEL
LIN {X 0,Y 545.097,Z 316.203,A -85,B 0,C 180,E1 -3711.496,E2 -3711.496} C_VEL
LIN {X 0,Y 545.216,Z 307.341,A -85,B 0,C 180,E1 -3714.362,E2 -3714.362} C_VEL
LIN {X 0,Y 545.334,Z 299.915,A -85,B 0,C 180,E1 -3716.812,E2 -3716.812} C_VEL
LIN {X 0,Y 545.481,Z 292.488,A -85,B 0,C 180,E1 -3719.314,E2 -3719.314} C_VEL
LIN {X 0,Y 545.666,Z 283.823,A -85,B 0,C 180,E1 -3722.311,E2 -3722.311} C_VEL
LIN {X 0,Y 545.797,Z 276.363,A -85,B 0,C 180,E1 -3724.961,E2 -3724.961} C_VEL
LIN {X 0,Y 545.989,Z 268.738,A -85,B 0,C 180,E1 -3727.693,E2 -3727.693} C_VEL
LIN {X 0,Y 546.094,Z 260.929,A -85,B 0,C 180,E1 -3730.597,E2 -3730.597} C_VEL
LIN {X 0,Y 545.965,Z 257.278,A -85,B 0,C 180,E1 -3732.019,E2 -3732.019} C_VEL
LIN {X 0,Y 545.089,Z 252.215,A -85,B 0,C 180,E1 -3734.3,E2 -3734.3} C_VEL
LIN {X 0,Y 545.067,Z 252.218,A -85,B 0,C 180,E1 -3737.303,E2 -3737.303} C_VEL
LIN {X 0,Y 545.07,Z 252.216,A -85,B 0,C 180,E1 -3739.857,E2 -3739.857} C_VEL
LIN {X 0,Y 545.075,Z 252.215,A -85,B 0,C 180,E1 -3743.074,E2 -3743.074} C_VEL
LIN {X 0,Y 545.055,Z 252.217,A -85,B 0,C 180,E1 -3746.327,E2 -3746.327} C_VEL
LIN {X 0,Y 545.072,Z 252.217,A -85,B 0,C 180,E1 -3748.952,E2 -3748.952} C_VEL
LIN {X 0,Y 545.09,Z 252.213,A -85,B 0,C 180,E1 -3751.507,E2 -3751.507} C_VEL
LIN {X 0,Y 545.1,Z 252.212,A -85,B 0,C 180,E1 -3754.491,E2 -3754.491} C_VEL
LIN {X 0,Y 545.043,Z 252.22,A -85,B 0,C 180,E1 -3757.242,E2 -3757.242} C_VEL
LIN {X 0,Y 545.127,Z 252.211,A -85,B 0,C 180,E1 -3760.415,E2 -3760.415} C_VEL
LIN {X 0,Y 545.078,Z 252.215,A -85,B 0,C 180,E1 -3763.521,E2 -3763.521} C_VEL
LIN {X 0,Y 545.098,Z 252.212,A -85,B 0,C 180,E1 -3765.819,E2 -3765.819} C_VEL
LIN {X 0,Y 545.122,Z 252.21,A -85,B 0,C 180,E1 -3768.849,E2 -3768.849} C_VEL
LIN {X 0,Y 545.133,Z 252.209,A -85,B 0,C 180,E1 -3771.846,E2 -3771.846} C_VEL
LIN {X 0,Y 545.205,Z 252.201,A -85,B 0,C 180,E1 -3774.822,E2 -3774.822} C_VEL
LIN {X 0,Y 545.199,Z 252.199,A -85,B 0,C 180,E1 -3777.783,E2 -3777.783} C_VEL
LIN {X 0,Y 545.218,Z 252.197,A -85,B 0,C 180,E1 -3780.738,E2 -3780.738} C_VEL
LIN {X 0,Y 545.175,Z 252.203,A -85,B 0,C 180,E1 -3782.955,E2 -3782.955} C_VEL
LIN {X 0,Y 545.171,Z 252.203,A -85,B 0,C 180,E1 -3785.919,E2 -3785.919} C_VEL
LIN {X 0,Y 545.119,Z 252.209,A -85,B 0,C 180,E1 -3788.899,E2 -3788.899} C_VEL
LIN {X 0,Y 545.138,Z 252.208,A -85,B 0,C 180,E1 -3791.903,E2 -3791.903} C_VEL
LIN {X 0,Y 545.088,Z 252.214,A -85,B 0,C 180,E1 -3794.943,E2 -3794.943} C_VEL
LIN {X 0,Y 545.082,Z 252.216,A -85,B 0,C 180,E1 -3798.025,E2 -3798.025} C_VEL
LIN {X 0,Y 545.093,Z 252.213,A -85,B 0,C 180,E1 -3800.371,E2 -3800.371} C_VEL
LIN {X 0,Y 545.092,Z 252.213,A -85,B 0,C 180,E1 -3803.558,E2 -3803.558} C_VEL
LIN {X 0,Y 545.08,Z 252.215,A -85,B 0,C 180,E1 -3805.999,E2 -3805.999} C_VEL
LIN {X 0,Y 545.09,Z 252.212,A -85,B 0,C 180,E1 -3808.747,E2 -3808.747} C_VEL
LIN {X 0,Y 545.057,Z 252.219,A -85,B 0,C 180,E1 -3811.678,E2 -3811.678} C_VEL
LIN {X 0,Y 545.08,Z 252.216,A -85,B 0,C 180,E1 -3814.562,E2 -3814.562} C_VEL
LIN {X 0,Y 545.063,Z 252.217,A -85,B 0,C 180,E1 -3817.005,E2 -3817.005} C_VEL
LIN {X 0,Y 544.355,Z 252.306,A -85,B 0,C 180,E1 -3817.622,E2 -3817.622} C_VEL
LIN {X 0,Y 541.491,Z 252.662,A -85,B 0,C 180,E1 -3818.622,E2 -3818.622} C_VEL
LIN {X 0,Y 539.105,Z 252.959,A -85,B 0,C 180,E1 -3819.428,E2 -3819.428} C_VEL
LIN {X 0,Y 538.095,Z 253.086,A -85,B 0,C 180,E1 -3820.05,E2 -3820.05} C_VEL
LIN {X 0,Y 538.018,Z 253.093,A -85,B 0,C 180,E1 -3820.261,E2 -3820.261} C_VEL
LIN {X 0,Y 538.029,Z 253.093,A -85,B 0,C 180,E1 -3822.987,E2 -3822.987} C_VEL
LIN {X 0,Y 538.025,Z 253.094,A -85,B 0,C 180,E1 -3825.924,E2 -3825.924} C_VEL
LIN {X 0,Y 538.073,Z 253.088,A -85,B 0,C 180,E1 -3829.248,E2 -3829.248} C_VEL
LIN {X 0,Y 537.988,Z 253.098,A -85,B 0,C 180,E1 -3832.121,E2 -3832.121} C_VEL
LIN {X 0,Y 538.013,Z 253.094,A -85,B 0,C 180,E1 -3834.916,E2 -3834.916} C_VEL
LIN {X 0,Y 538.025,Z 253.095,A -85,B 0,C 180,E1 -3837.617,E2 -3837.617} C_VEL
LIN {X 0,Y 538.036,Z 253.091,A -85,B 0,C 180,E1 -3840.239,E2 -3840.239} C_VEL
LIN {X 0,Y 538.064,Z 253.088,A -85,B 0,C 180,E1 -3842.796,E2 -3842.796} C_VEL
LIN {X 0,Y 538.041,Z 253.092,A -85,B 0,C 180,E1 -3845.292,E2 -3845.292} C_VEL
LIN {X 0,Y 538.006,Z 253.097,A -85,B 0,C 180,E1 -3848.041,E2 -3848.041} C_VEL
LIN {X 0,Y 538.032,Z 253.092,A -85,B 0,C 180,E1 -3850.939,E2 -3850.939} C_VEL
LIN {X 0,Y 538.018,Z 253.096,A -85,B 0,C 180,E1 -3853.298,E2 -3853.298} C_VEL
LIN {X 0,Y 538.054,Z 253.09,A -85,B 0,C 180,E1 -3855.63,E2 -3855.63} C_VEL
LIN {X 0,Y 538.08,Z 253.087,A -85,B 0,C 180,E1 -3858.701,E2 -3858.701} C_VEL
LIN {X 0,Y 538.083,Z 253.087,A -85,B 0,C 180,E1 -3861.739,E2 -3861.739} C_VEL
LIN {X 0,Y 538.116,Z 253.081,A -85,B 0,C 180,E1 -3864.002,E2 -3864.002} C_VEL
LIN {X 0,Y 537.833,Z 253.12,A -85,B 0,C 180,E1 -3866.253,E2 -3866.253} C_VEL
LIN {X 0,Y 537.74,Z 253.133,A -85,B 0,C 180,E1 -3867.003,E2 -3867.003} C_VEL
LIN {X 0,Y 537.956,Z 255.294,A -85,B 0,C 180,E1 -3869.251,E2 -3869.251} C_VEL
LIN {X 0,Y 537.766,Z 257.485,A -85,B 0,C 180,E1 -3871.497,E2 -3871.497} C_VEL
LIN {X 0,Y 537.695,Z 260.408,A -85,B 0,C 180,E1 -3874.497,E2 -3874.497} C_VEL
LIN {X 0,Y 537.679,Z 263.325,A -85,B 0,C 180,E1 -3877.51,E2 -3877.51} C_VEL
LIN {X 0,Y 537.633,Z 266.28,A -85,B 0,C 180,E1 -3880.545,E2 -3880.545} C_VEL
LIN {X 0,Y 537.521,Z 269.271,A -85,B 0,C 180,E1 -3883.611,E2 -3883.611} C_VEL
LIN {X 0,Y 537.56,Z 269.895,A -85,B 0,C 180,E1 -3884.262,E2 -3884.262} C_VEL
LIN {X 0,Y 540.901,Z 283.879,A -85,B 0,C 180,E1 -3884.66,E2 -3884.66} C_VEL
LIN {X 0,Y 540.588,Z 299.494,A -85,B 0,C 180,E1 -3885.109,E2 -3885.109} C_VEL
LIN {X 0,Y 540.199,Z 314.217,A -85,B 0,C 180,E1 -3885.695,E2 -3885.695} C_VEL
LIN {X 0,Y 539.825,Z 327.052,A -85,B 0,C 180,E1 -3886.351,E2 -3886.351} C_VEL
LIN {X 0,Y 539.451,Z 341.12,A -85,B 0,C 180,E1 -3887.24,E2 -3887.24} C_VEL
LIN {X 0,Y 539.077,Z 354.02,A -85,B 0,C 180,E1 -3888.233,E2 -3888.233} C_VEL
LIN {X 0,Y 538.694,Z 364.896,A -85,B 0,C 180,E1 -3889.233,E2 -3889.233} C_VEL
LIN {X 0,Y 538.401,Z 376.117,A -85,B 0,C 180,E1 -3890.457,E2 -3890.457} C_VEL
LIN {X 0,Y 538.117,Z 385.767,A -85,B 0,C 180,E1 -3891.712,E2 -3891.712} C_VEL
LIN {X 0,Y 537.914,Z 394.526,A -85,B 0,C 180,E1 -3893.076,E2 -3893.076} C_VEL
LIN {X 0,Y 537.753,Z 401.175,A -85,B 0,C 180,E1 -3894.31,E2 -3894.31} C_VEL
LIN {X 0,Y 537.677,Z 406.956,A -85,B 0,C 180,E1 -3895.594,E2 -3895.594} C_VEL
LIN {X 0,Y 537.561,Z 411.404,A -85,B 0,C 180,E1 -3896.81,E2 -3896.81} C_VEL
LIN {X 0,Y 537.514,Z 415.179,A -85,B 0,C 180,E1 -3898.079,E2 -3898.079} C_VEL
LIN {X 0,Y 537.495,Z 417.181,A -85,B 0,C 180,E1 -3898.933,E2 -3898.933} C_VEL
LIN {X 0,Y 537.492,Z 419.633,A -85,B 0,C 180,E1 -3900.349,E2 -3900.349} C_VEL
LIN {X 0,Y 537.442,Z 421.065,A -85,B 0,C 180,E1 -3901.792,E2 -3901.792} C_VEL
LIN {X 0,Y 537.451,Z 421.45,A -85,B 0,C 180,E1 -3903.312,E2 -3903.312} C_VEL
LIN {X 0,Y 537.457,Z 420.915,A -85,B 0,C 180,E1 -3904.534,E2 -3904.534} C_VEL
LIN {X 0,Y 537.441,Z 419.18,A -85,B 0,C 180,E1 -3906.047,E2 -3906.047} C_VEL
LIN {X 0,Y 537.473,Z 417.3,A -85,B 0,C 180,E1 -3907.097,E2 -3907.097} C_VEL
LIN {X 0,Y 537.555,Z 414.28,A -85,B 0,C 180,E1 -3908.333,E2 -3908.333} C_VEL
LIN {X 0,Y 537.613,Z 409.489,A -85,B 0,C 180,E1 -3909.833,E2 -3909.833} C_VEL
LIN {X 0,Y 537.681,Z 403.454,A -85,B 0,C 180,E1 -3911.305,E2 -3911.305} C_VEL
LIN {X 0,Y 537.86,Z 395.79,A -85,B 0,C 180,E1 -3912.801,E2 -3912.801} C_VEL
LIN {X 0,Y 538.114,Z 386.855,A -85,B 0,C 180,E1 -3914.224,E2 -3914.224} C_VEL
LIN {X 0,Y 538.367,Z 377.331,A -85,B 0,C 180,E1 -3915.491,E2 -3915.491} C_VEL
LIN {X 0,Y 538.688,Z 366.083,A -85,B 0,C 180,E1 -3916.74,E2 -3916.74} C_VEL
LIN {X 0,Y 539.073,Z 353.849,A -85,B 0,C 180,E1 -3917.871,E2 -3917.871} C_VEL
LIN {X 0,Y 539.525,Z 341.105,A -85,B 0,C 180,E1 -3918.848,E2 -3918.848} C_VEL
LIN {X 0,Y 539.886,Z 327.725,A -85,B 0,C 180,E1 -3919.7,E2 -3919.7} C_VEL
LIN {X 0,Y 540.298,Z 313.939,A -85,B 0,C 180,E1 -3920.405,E2 -3920.405} C_VEL
LIN {X 0,Y 540.602,Z 299.13,A -85,B 0,C 180,E1 -3920.994,E2 -3920.994} C_VEL
LIN {X 0,Y 540.885,Z 283.758,A -85,B 0,C 180,E1 -3921.434,E2 -3921.434} C_VEL
LIN {X 0,Y 537.892,Z 271.612,A -85,B 0,C 180,E1 -3921.781,E2 -3921.781} C_VEL
LIN {X 0,Y 537.547,Z 269.95,A -85,B 0,C 180,E1 -3921.841,E2 -3921.841} C_VEL
LIN {X 0,Y 537.592,Z 267.098,A -85,B 0,C 180,E1 -3924.887,E2 -3924.887} C_VEL
LIN {X 0,Y 537.662,Z 264.672,A -85,B 0,C 180,E1 -3927.595,E2 -3927.595} C_VEL
LIN {X 0,Y 537.712,Z 262.239,A -85,B 0,C 180,E1 -3930.222,E2 -3930.222} C_VEL
LIN {X 0,Y 537.736,Z 259.856,A -85,B 0,C 180,E1 -3932.779,E2 -3932.779} C_VEL
LIN {X 0,Y 537.804,Z 257.505,A -85,B 0,C 180,E1 -3935.282,E2 -3935.282} C_VEL
LIN {X 0,Y 537.831,Z 254.833,A -85,B 0,C 180,E1 -3938.089,E2 -3938.089} C_VEL
LIN {X 0,Y 537.854,Z 253.118,A -85,B 0,C 180,E1 -3940.185,E2 -3940.185} C_VEL
LIN {X 0,Y 538.019,Z 253.097,A -85,B 0,C 180,E1 -3942.517,E2 -3942.517} C_VEL
LIN {X 0,Y 538.058,Z 253.091,A -85,B 0,C 180,E1 -3945.632,E2 -3945.632} C_VEL
LIN {X 0,Y 538.071,Z 253.089,A -85,B 0,C 180,E1 -3948.702,E2 -3948.702} C_VEL
LIN {X 0,Y 538.083,Z 253.087,A -85,B 0,C 180,E1 -3951.74,E2 -3951.74} C_VEL
LIN {X 0,Y 538.16,Z 253.076,A -85,B 0,C 180,E1 -3954.756,E2 -3954.756} C_VEL
LIN {X 0,Y 538.166,Z 253.075,A -85,B 0,C 180,E1 -3957.756,E2 -3957.756} C_VEL
LIN {X 0,Y 538.18,Z 253.074,A -85,B 0,C 180,E1 -3960.749,E2 -3960.749} C_VEL
LIN {X 0,Y 538.138,Z 253.079,A -85,B 0,C 180,E1 -3962.995,E2 -3962.995} C_VEL
LIN {X 0,Y 538.121,Z 253.08,A -85,B 0,C 180,E1 -3965.998,E2 -3965.998} C_VEL
LIN {X 0,Y 538.07,Z 253.088,A -85,B 0,C 180,E1 -3969.018,E2 -3969.018} C_VEL
LIN {X 0,Y 538.081,Z 253.087,A -85,B 0,C 180,E1 -3972.063,E2 -3972.063} C_VEL
LIN {X 0,Y 538.043,Z 253.092,A -85,B 0,C 180,E1 -3975.144,E2 -3975.144} C_VEL
LIN {X 0,Y 538.028,Z 253.094,A -85,B 0,C 180,E1 -3978.271,E2 -3978.271} C_VEL
LIN {X 0,Y 538.04,Z 253.092,A -85,B 0,C 180,E1 -3980.652,E2 -3980.652} C_VEL
LIN {X 0,Y 538.022,Z 253.094,A -85,B 0,C 180,E1 -3983.888,E2 -3983.888} C_VEL
LIN {X 0,Y 538.048,Z 253.091,A -85,B 0,C 180,E1 -3986.367,E2 -3986.367} C_VEL
LIN {X 0,Y 538.028,Z 253.095,A -85,B 0,C 180,E1 -3988.934,E2 -3988.934} C_VEL
LIN {X 0,Y 538.008,Z 253.099,A -85,B 0,C 180,E1 -3991.888,E2 -3991.888} C_VEL
LIN {X 0,Y 538.011,Z 253.098,A -85,B 0,C 180,E1 -3994.618,E2 -3994.618} C_VEL
LIN {X 0,Y 538.003,Z 253.099,A -85,B 0,C 180,E1 -3997.171,E2 -3997.171} C_VEL
LIN {X 0,Y 538.028,Z 253.095,A -85,B 0,C 180,E1 -3999.797,E2 -3999.797} C_VEL
LIN {X 0,Y 538.017,Z 253.097,A -85,B 0,C 180,E1 -4002.787,E2 -4002.787} C_VEL
LIN {X 0,Y 538.039,Z 253.268,A -85,B 0,C 180,E1 -4005.605,E2 -4005.605} C_VEL
LIN {X 0,Y 539.026,Z 258.803,A -85,B 0,C 180,E1 -4008.004,E2 -4008.004} C_VEL
LIN {X 0,Y 539.087,Z 264.408,A -85,B 0,C 180,E1 -4010.28,E2 -4010.28} C_VEL
LIN {X 0,Y 538.898,Z 272.202,A -85,B 0,C 180,E1 -4013.138,E2 -4013.138} C_VEL
LIN {X 0,Y 538.762,Z 280.077,A -85,B 0,C 180,E1 -4015.881,E2 -4015.881} C_VEL
LIN {X 0,Y 538.584,Z 287.54,A -85,B 0,C 180,E1 -4018.537,E2 -4018.537} C_VEL
LIN {X 0,Y 538.455,Z 294.967,A -85,B 0,C 180,E1 -4021.124,E2 -4021.124} C_VEL
LIN {X 0,Y 538.277,Z 304.267,A -85,B 0,C 180,E1 -4024.276,E2 -4024.276} C_VEL
LIN {X 0,Y 538.079,Z 313.534,A -85,B 0,C 180,E1 -4027.338,E2 -4027.338} C_VEL
LIN {X 0,Y 537.978,Z 322.218,A -85,B 0,C 180,E1 -4030.151,E2 -4030.151} C_VEL
LIN {X 0,Y 537.908,Z 325.422,A -85,B 0,C 180,E1 -4031.175,E2 -4031.175} C_VEL
LIN {X 0,Y 540.953,Z 338.68,A -85,B 0,C 180,E1 -4031.509,E2 -4031.509} C_VEL
LIN {X 0,Y 540.7,Z 353.714,A -85,B 0,C 180,E1 -4031.887,E2 -4031.887} C_VEL
LIN {X 0,Y 540.396,Z 369.014,A -85,B 0,C 180,E1 -4032.436,E2 -4032.436} C_VEL
LIN {X 0,Y 540.018,Z 382.614,A -85,B 0,C 180,E1 -4033.071,E2 -4033.071} C_VEL
LIN {X 0,Y 539.657,Z 395.787,A -85,B 0,C 180,E1 -4033.838,E2 -4033.838} C_VEL
LIN {X 0,Y 539.267,Z 409.522,A -85,B 0,C 180,E1 -4034.822,E2 -4034.822} C_VEL
LIN {X 0,Y 538.85,Z 421.388,A -85,B 0,C 180,E1 -4035.845,E2 -4035.845} C_VEL
LIN {X 0,Y 538.525,Z 432.514,A -85,B 0,C 180,E1 -4036.991,E2 -4036.991} C_VEL
LIN {X 0,Y 538.178,Z 442.734,A -85,B 0,C 180,E1 -4038.243,E2 -4038.243} C_VEL
LIN {X 0,Y 538.017,Z 452.297,A -85,B 0,C 180,E1 -4039.653,E2 -4039.653} C_VEL
LIN {X 0,Y 537.797,Z 459.754,A -85,B 0,C 180,E1 -4040.978,E2 -4040.978} C_VEL
LIN {X 0,Y 537.661,Z 466.704,A -85,B 0,C 180,E1 -4042.49,E2 -4042.49} C_VEL
LIN {X 0,Y 537.623,Z 472.164,A -85,B 0,C 180,E1 -4043.998,E2 -4043.998} C_VEL
LIN {X 0,Y 537.508,Z 476.292,A -85,B 0,C 180,E1 -4045.501,E2 -4045.501} C_VEL
LIN {X 0,Y 537.544,Z 479.188,A -85,B 0,C 180,E1 -4047.003,E2 -4047.003} C_VEL
LIN {X 0,Y 537.449,Z 480.911,A -85,B 0,C 180,E1 -4048.502,E2 -4048.502} C_VEL
LIN {X 0,Y 537.439,Z 481.5,A -85,B 0,C 180,E1 -4050.001,E2 -4050.001} C_VEL
LIN {X 0,Y 537.449,Z 480.91,A -85,B 0,C 180,E1 -4051.499,E2 -4051.499} C_VEL
LIN {X 0,Y 537.544,Z 479.184,A -85,B 0,C 180,E1 -4052.998,E2 -4052.998} C_VEL
LIN {X 0,Y 537.508,Z 476.288,A -85,B 0,C 180,E1 -4054.5,E2 -4054.5} C_VEL
LIN {X 0,Y 537.62,Z 472.162,A -85,B 0,C 180,E1 -4056.003,E2 -4056.003} C_VEL
LIN {X 0,Y 537.662,Z 466.7,A -85,B 0,C 180,E1 -4057.511,E2 -4057.511} C_VEL
LIN {X 0,Y 537.798,Z 459.745,A -85,B 0,C 180,E1 -4059.023,E2 -4059.023} C_VEL
LIN {X 0,Y 538.024,Z 451.084,A -85,B 0,C 180,E1 -4060.538,E2 -4060.538} C_VEL
LIN {X 0,Y 538.23,Z 441.532,A -85,B 0,C 180,E1 -4061.912,E2 -4061.912} C_VEL
LIN {X 0,Y 538.525,Z 432.504,A -85,B 0,C 180,E1 -4063.01,E2 -4063.01} C_VEL
LIN {X 0,Y 538.842,Z 421.38,A -85,B 0,C 180,E1 -4064.156,E2 -4064.156} C_VEL
LIN {X 0,Y 539.235,Z 409.582,A -85,B 0,C 180,E1 -4065.174,E2 -4065.174} C_VEL
LIN {X 0,Y 539.618,Z 395.77,A -85,B 0,C 180,E1 -4066.165,E2 -4066.165} C_VEL
LIN {X 0,Y 540.013,Z 382.591,A -85,B 0,C 180,E1 -4066.93,E2 -4066.93} C_VEL
LIN {X 0,Y 540.38,Z 369.006,A -85,B 0,C 180,E1 -4067.565,E2 -4067.565} C_VEL
LIN {X 0,Y 540.696,Z 354.409,A -85,B 0,C 180,E1 -4068.091,E2 -4068.091} C_VEL
LIN {X 0,Y 540.925,Z 340.117,A -85,B 0,C 180,E1 -4068.461,E2 -4068.461} C_VEL
LIN {X 0,Y 540.65,Z 336.795,A -85,B 0,C 180,E1 -4068.542,E2 -4068.542} C_VEL
LIN {X 0,Y 537.908,Z 325.356,A -85,B 0,C 180,E1 -4068.846,E2 -4068.846} C_VEL
LIN {X 0,Y 538.056,Z 317.244,A -85,B 0,C 180,E1 -4071.453,E2 -4071.453} C_VEL
LIN {X 0,Y 538.183,Z 308.581,A -85,B 0,C 180,E1 -4074.29,E2 -4074.29} C_VEL
LIN {X 0,Y 538.347,Z 299.915,A -85,B 0,C 180,E1 -4077.189,E2 -4077.189} C_VEL
LIN {X 0,Y 538.532,Z 291.327,A -85,B 0,C 180,E1 -4080.135,E2 -4080.135} C_VEL
LIN {X 0,Y 538.729,Z 282.585,A -85,B 0,C 180,E1 -4083.224,E2 -4083.224} C_VEL
LIN {X 0,Y 538.93,Z 273.673,A -85,B 0,C 180,E1 -4086.41,E2 -4086.41} C_VEL
LIN {X 0,Y 539.109,Z 266.076,A -85,B 0,C 180,E1 -4089.218,E2 -4089.218} C_VEL
LIN {X 0,Y 539.122,Z 259.692,A -85,B 0,C 180,E1 -4091.67,E2 -4091.67} C_VEL
LIN {X 0,Y 538.241,Z 254.128,A -85,B 0,C 180,E1 -4094.097,E2 -4094.097} C_VEL
LIN {X 0,Y 538.032,Z 253.094,A -85,B 0,C 180,E1 -4094.609,E2 -4094.609} C_VEL
LIN {X 0,Y 538.024,Z 253.095,A -85,B 0,C 180,E1 -4097.214,E2 -4097.214} C_VEL
LIN {X 0,Y 538.028,Z 253.094,A -85,B 0,C 180,E1 -4100.203,E2 -4100.203} C_VEL
LIN {X 0,Y 538.029,Z 253.092,A -85,B 0,C 180,E1 -4103.067,E2 -4103.067} C_VEL
LIN {X 0,Y 538.016,Z 253.095,A -85,B 0,C 180,E1 -4105.826,E2 -4105.826} C_VEL
LIN {X 0,Y 538.014,Z 253.095,A -85,B 0,C 180,E1 -4108.498,E2 -4108.498} C_VEL
LIN {X 0,Y 538.025,Z 253.094,A -85,B 0,C 180,E1 -4111.097,E2 -4111.097} C_VEL
LIN {X 0,Y 538.047,Z 253.09,A -85,B 0,C 180,E1 -4113.633,E2 -4113.633} C_VEL
LIN {X 0,Y 538.013,Z 253.095,A -85,B 0,C 180,E1 -4116.122,E2 -4116.122} C_VEL
LIN {X 0,Y 538.045,Z 253.091,A -85,B 0,C 180,E1 -4119.348,E2 -4119.348} C_VEL
LIN {X 0,Y 538.061,Z 253.091,A -85,B 0,C 180,E1 -4122.517,E2 -4122.517} C_VEL
LIN {X 0,Y 538.068,Z 253.088,A -85,B 0,C 180,E1 -4125.63,E2 -4125.63} C_VEL
LIN {X 0,Y 538.082,Z 253.088,A -85,B 0,C 180,E1 -4128.701,E2 -4128.701} C_VEL
LIN {X 0,Y 538.089,Z 253.085,A -85,B 0,C 180,E1 -4131.739,E2 -4131.739} C_VEL
LIN {X 0,Y 538.162,Z 253.077,A -85,B 0,C 180,E1 -4134.754,E2 -4134.754} C_VEL
LIN {X 0,Y 538.171,Z 253.074,A -85,B 0,C 180,E1 -4137.754,E2 -4137.754} C_VEL
LIN {X 0,Y 538.188,Z 253.073,A -85,B 0,C 180,E1 -4140.747,E2 -4140.747} C_VEL
LIN {X 0,Y 538.142,Z 253.079,A -85,B 0,C 180,E1 -4142.994,E2 -4142.994} C_VEL
LIN {X 0,Y 538.125,Z 253.081,A -85,B 0,C 180,E1 -4145.996,E2 -4145.996} C_VEL
LIN {X 0,Y 538.07,Z 253.087,A -85,B 0,C 180,E1 -4149.017,E2 -4149.017} C_VEL
LIN {X 0,Y 538.086,Z 253.086,A -85,B 0,C 180,E1 -4152.061,E2 -4152.061} C_VEL
LIN {X 0,Y 538.048,Z 253.09,A -85,B 0,C 180,E1 -4155.143,E2 -4155.143} C_VEL
LIN {X 0,Y 538.034,Z 253.093,A -85,B 0,C 180,E1 -4158.269,E2 -4158.269} C_VEL
LIN {X 0,Y 538.038,Z 253.092,A -85,B 0,C 180,E1 -4160.65,E2 -4160.65} C_VEL
LIN {X 0,Y 538.025,Z 253.093,A -85,B 0,C 180,E1 -4163.886,E2 -4163.886} C_VEL
LIN {X 0,Y 538.042,Z 253.092,A -85,B 0,C 180,E1 -4166.365,E2 -4166.365} C_VEL
LIN {X 0,Y 538.031,Z 253.091,A -85,B 0,C 180,E1 -4168.933,E2 -4168.933} C_VEL
LIN {X 0,Y 538.013,Z 253.095,A -85,B 0,C 180,E1 -4171.887,E2 -4171.887} C_VEL
LIN {X 0,Y 538.03,Z 253.094,A -85,B 0,C 180,E1 -4174.62,E2 -4174.62} C_VEL
LIN {X 0,Y 538.005,Z 253.095,A -85,B 0,C 180,E1 -4177.169,E2 -4177.169} C_VEL
LIN {X 0,Y 538.018,Z 253.093,A -85,B 0,C 180,E1 -4180.261,E2 -4180.261} C_VEL
LIN {X 0,Y 537.368,Z 253.176,A -85,B 0,C 180,E1 -4180.886,E2 -4180.886} C_VEL
LIN {X 0,Y 534.518,Z 253.533,A -85,B 0,C 180,E1 -4181.901,E2 -4181.901} C_VEL
LIN {X 0,Y 532.095,Z 253.835,A -85,B 0,C 180,E1 -4182.718,E2 -4182.718} C_VEL
LIN {X 0,Y 531.047,Z 253.963,A -85,B 0,C 180,E1 -4183.349,E2 -4183.349} C_VEL
LIN {X 0,Y 530.959,Z 253.973,A -85,B 0,C 180,E1 -4183.563,E2 -4183.563} C_VEL
LIN {X 0,Y 530.962,Z 253.972,A -85,B 0,C 180,E1 -4186.505,E2 -4186.505} C_VEL
LIN {X 0,Y 531.021,Z 253.967,A -85,B 0,C 180,E1 -4189.57,E2 -4189.57} C_VEL
LIN {X 0,Y 530.964,Z 253.973,A -85,B 0,C 180,E1 -4192.575,E2 -4192.575} C_VEL
LIN {X 0,Y 530.994,Z 253.969,A -85,B 0,C 180,E1 -4195.31,E2 -4195.31} C_VEL
LIN {X 0,Y 530.976,Z 253.971,A -85,B 0,C 180,E1 -4198.032,E2 -4198.032} C_VEL
LIN {X 0,Y 530.999,Z 253.969,A -85,B 0,C 180,E1 -4200.869,E2 -4200.869} C_VEL
LIN {X 0,Y 531.004,Z 253.968,A -85,B 0,C 180,E1 -4203.256,E2 -4203.256} C_VEL
LIN {X 0,Y 530.988,Z 253.972,A -85,B 0,C 180,E1 -4205.957,E2 -4205.957} C_VEL
LIN {X 0,Y 530.993,Z 253.969,A -85,B 0,C 180,E1 -4209.061,E2 -4209.061} C_VEL
LIN {X 0,Y 531.007,Z 253.968,A -85,B 0,C 180,E1 -4212.277,E2 -4212.277} C_VEL
LIN {X 0,Y 531.031,Z 253.967,A -85,B 0,C 180,E1 -4215.436,E2 -4215.436} C_VEL
LIN {X 0,Y 531.037,Z 253.964,A -85,B 0,C 180,E1 -4218.549,E2 -4218.549} C_VEL
LIN {X 0,Y 531.052,Z 253.964,A -85,B 0,C 180,E1 -4221.629,E2 -4221.629} C_VEL
LIN {X 0,Y 531.082,Z 253.957,A -85,B 0,C 180,E1 -4224.684,E2 -4224.684} C_VEL
LIN {X 0,Y 530.698,Z 254.01,A -85,B 0,C 180,E1 -4226.963,E2 -4226.963} C_VEL
LIN {X 0,Y 530.915,Z 255.963,A -85,B 0,C 180,E1 -4229.241,E2 -4229.241} C_VEL
LIN {X 0,Y 530.692,Z 258.193,A -85,B 0,C 180,E1 -4231.517,E2 -4231.517} C_VEL
LIN {X 0,Y 530.636,Z 261.129,A -85,B 0,C 180,E1 -4234.557,E2 -4234.557} C_VEL
LIN {X 0,Y 530.595,Z 264.082,A -85,B 0,C 180,E1 -4237.611,E2 -4237.611} C_VEL
LIN {X 0,Y 530.555,Z 267.068,A -85,B 0,C 180,E1 -4240.687,E2 -4240.687} C_VEL
LIN {X 0,Y 530.481,Z 270.089,A -85,B 0,C 180,E1 -4243.796,E2 -4243.796} C_VEL
LIN {X 0,Y 530.505,Z 270.473,A -85,B 0,C 180,E1 -4244.015,E2 -4244.015} C_VEL
LIN {X 0,Y 534.172,Z 284.486,A -85,B 0,C 180,E1 -4244.427,E2 -4244.427} C_VEL
LIN {X 0,Y 533.835,Z 299.357,A -85,B 0,C 180,E1 -4244.858,E2 -4244.858} C_VEL
LIN {X 0,Y 533.44,Z 314.286,A -85,B 0,C 180,E1 -4245.456,E2 -4245.456} C_VEL
LIN {X 0,Y 533.022,Z 328.12,A -85,B 0,C 180,E1 -4246.172,E2 -4246.172} C_VEL
LIN {X 0,Y 532.607,Z 342.055,A -85,B 0,C 180,E1 -4247.073,E2 -4247.073} C_VEL
LIN {X 0,Y 532.188,Z 354.406,A -85,B 0,C 180,E1 -4248.048,E2 -4248.048} C_VEL
LIN {X 0,Y 531.743,Z 365.488,A -85,B 0,C 180,E1 -4249.093,E2 -4249.093} C_VEL
LIN {X 0,Y 531.409,Z 376.182,A -85,B 0,C 180,E1 -4250.293,E2 -4250.293} C_VEL
LIN {X 0,Y 531.083,Z 385.651,A -85,B 0,C 180,E1 -4251.544,E2 -4251.544} C_VEL
LIN {X 0,Y 530.862,Z 394.79,A -85,B 0,C 180,E1 -4252.988,E2 -4252.988} C_VEL
LIN {X 0,Y 530.697,Z 401.386,A -85,B 0,C 180,E1 -4254.238,E2 -4254.238} C_VEL
LIN {X 0,Y 530.567,Z 407.932,A -85,B 0,C 180,E1 -4255.748,E2 -4255.748} C_VEL
LIN {X 0,Y 530.484,Z 412.61,A -85,B 0,C 180,E1 -4257.098,E2 -4257.098} C_VEL
LIN {X 0,Y 530.415,Z 416.297,A -85,B 0,C 180,E1 -4258.489,E2 -4258.489} C_VEL
LIN {X 0,Y 530.411,Z 419.511,A -85,B 0,C 180,E1 -4260.231,E2 -4260.231} C_VEL
LIN {X 0,Y 530.362,Z 421.212,A -85,B 0,C 180,E1 -4262.008,E2 -4262.008} C_VEL
LIN {X 0,Y 530.346,Z 421.432,A -85,B 0,C 180,E1 -4263.402,E2 -4263.402} C_VEL
LIN {X 0,Y 530.363,Z 420.776,A -85,B 0,C 180,E1 -4264.759,E2 -4264.759} C_VEL
LIN {X 0,Y 530.342,Z 419.209,A -85,B 0,C 180,E1 -4266.066,E2 -4266.066} C_VEL
LIN {X 0,Y 530.388,Z 416.408,A -85,B 0,C 180,E1 -4267.555,E2 -4267.555} C_VEL
LIN {X 0,Y 530.49,Z 412.551,A -85,B 0,C 180,E1 -4269.009,E2 -4269.009} C_VEL
LIN {X 0,Y 530.56,Z 407.452,A -85,B 0,C 180,E1 -4270.471,E2 -4270.471} C_VEL
LIN {X 0,Y 530.695,Z 400.04,A -85,B 0,C 180,E1 -4272.133,E2 -4272.133} C_VEL
LIN {X 0,Y 530.933,Z 392.501,A -85,B 0,C 180,E1 -4273.497,E2 -4273.497} C_VEL
LIN {X 0,Y 531.128,Z 383.886,A -85,B 0,C 180,E1 -4274.798,E2 -4274.798} C_VEL
LIN {X 0,Y 531.47,Z 373.59,A -85,B 0,C 180,E1 -4276.111,E2 -4276.111} C_VEL
LIN {X 0,Y 531.924,Z 362.108,A -85,B 0,C 180,E1 -4277.335,E2 -4277.335} C_VEL
LIN {X 0,Y 532.313,Z 351.178,A -85,B 0,C 180,E1 -4278.313,E2 -4278.313} C_VEL
LIN {X 0,Y 532.761,Z 338.91,A -85,B 0,C 180,E1 -4279.235,E2 -4279.235} C_VEL
LIN {X 0,Y 533.156,Z 325.305,A -85,B 0,C 180,E1 -4280.076,E2 -4280.076} C_VEL
LIN {X 0,Y 533.609,Z 310.718,A -85,B 0,C 180,E1 -4280.79,E2 -4280.79} C_VEL
LIN {X 0,Y 533.944,Z 295.741,A -85,B 0,C 180,E1 -4281.349,E2 -4281.349} C_VEL
LIN {X 0,Y 534.038,Z 284.017,A -85,B 0,C 180,E1 -4281.68,E2 -4281.68} C_VEL
LIN {X 0,Y 531.036,Z 272.628,A -85,B 0,C 180,E1 -4282.02,E2 -4282.02} C_VEL
LIN {X 0,Y 530.485,Z 270.467,A -85,B 0,C 180,E1 -4282.094,E2 -4282.094} C_VEL
LIN {X 0,Y 530.548,Z 267.541,A -85,B 0,C 180,E1 -4285.279,E2 -4285.279} C_VEL
LIN {X 0,Y 530.622,Z 265.028,A -85,B 0,C 180,E1 -4288.01,E2 -4288.01} C_VEL
LIN {X 0,Y 530.663,Z 262.308,A -85,B 0,C 180,E1 -4290.936,E2 -4290.936} C_VEL
LIN {X 0,Y 530.697,Z 259.398,A -85,B 0,C 180,E1 -4294.087,E2 -4294.087} C_VEL
LIN {X 0,Y 530.744,Z 257.05,A -85,B 0,C 180,E1 -4296.595,E2 -4296.595} C_VEL
LIN {X 0,Y 530.741,Z 254.714,A -85,B 0,C 180,E1 -4299.053,E2 -4299.053} C_VEL
LIN {X 0,Y 530.81,Z 253.995,A -85,B 0,C 180,E1 -4300.058,E2 -4300.058} C_VEL
LIN {X 0,Y 530.974,Z 253.975,A -85,B 0,C 180,E1 -4302.361,E2 -4302.361} C_VEL
LIN {X 0,Y 531.013,Z 253.969,A -85,B 0,C 180,E1 -4305.437,E2 -4305.437} C_VEL
LIN {X 0,Y 531.031,Z 253.965,A -85,B 0,C 180,E1 -4308.551,E2 -4308.551} C_VEL
LIN {X 0,Y 531.052,Z 253.962,A -85,B 0,C 180,E1 -4311.63,E2 -4311.63} C_VEL
LIN {X 0,Y 531.119,Z 253.953,A -85,B 0,C 180,E1 -4314.686,E2 -4314.686} C_VEL
LIN {X 0,Y 531.137,Z 253.95,A -85,B 0,C 180,E1 -4317.726,E2 -4317.726} C_VEL
LIN {X 0,Y 531.15,Z 253.95,A -85,B 0,C 180,E1 -4320.759,E2 -4320.759} C_VEL
LIN {X 0,Y 531.104,Z 253.955,A -85,B 0,C 180,E1 -4323.035,E2 -4323.035} C_VEL
LIN {X 0,Y 531.081,Z 253.957,A -85,B 0,C 180,E1 -4326.078,E2 -4326.078} C_VEL
LIN {X 0,Y 531.031,Z 253.965,A -85,B 0,C 180,E1 -4329.139,E2 -4329.139} C_VEL
LIN {X 0,Y 531.038,Z 253.963,A -85,B 0,C 180,E1 -4332.226,E2 -4332.226} C_VEL
LIN {X 0,Y 530.993,Z 253.969,A -85,B 0,C 180,E1 -4335.35,E2 -4335.35} C_VEL
LIN {X 0,Y 530.987,Z 253.97,A -85,B 0,C 180,E1 -4338.522,E2 -4338.522} C_VEL
LIN {X 0,Y 531,Z 253.968,A -85,B 0,C 180,E1 -4340.938,E2 -4340.938} C_VEL
LIN {X 0,Y 530.978,Z 253.971,A -85,B 0,C 180,E1 -4344.225,E2 -4344.225} C_VEL
LIN {X 0,Y 531.009,Z 253.969,A -85,B 0,C 180,E1 -4346.744,E2 -4346.744} C_VEL
LIN {X 0,Y 530.979,Z 253.972,A -85,B 0,C 180,E1 -4349.323,E2 -4349.323} C_VEL
LIN {X 0,Y 530.963,Z 253.976,A -85,B 0,C 180,E1 -4352.101,E2 -4352.101} C_VEL
LIN {X 0,Y 530.969,Z 253.976,A -85,B 0,C 180,E1 -4354.852,E2 -4354.852} C_VEL
LIN {X 0,Y 530.964,Z 253.977,A -85,B 0,C 180,E1 -4357.508,E2 -4357.508} C_VEL
LIN {X 0,Y 530.983,Z 253.972,A -85,B 0,C 180,E1 -4360.433,E2 -4360.433} C_VEL
LIN {X 0,Y 530.963,Z 253.975,A -85,B 0,C 180,E1 -4363.495,E2 -4363.495} C_VEL
LIN {X 0,Y 530.997,Z 254.046,A -85,B 0,C 180,E1 -4365.241,E2 -4365.241} C_VEL
LIN {X 0,Y 531.956,Z 259.573,A -85,B 0,C 180,E1 -4367.719,E2 -4367.719} C_VEL
LIN {X 0,Y 532.189,Z 264.39,A -85,B 0,C 180,E1 -4369.679,E2 -4369.679} C_VEL
LIN {X 0,Y 531.958,Z 271.502,A -85,B 0,C 180,E1 -4372.438,E2 -4372.438} C_VEL
LIN {X 0,Y 531.779,Z 279.765,A -85,B 0,C 180,E1 -4375.37,E2 -4375.37} C_VEL
LIN {X 0,Y 531.642,Z 287.54,A -85,B 0,C 180,E1 -4378.078,E2 -4378.078} C_VEL
LIN {X 0,Y 531.467,Z 296.303,A -85,B 0,C 180,E1 -4381.175,E2 -4381.175} C_VEL
LIN {X 0,Y 531.285,Z 304.869,A -85,B 0,C 180,E1 -4384.118,E2 -4384.118} C_VEL
LIN {X 0,Y 531.06,Z 313.534,A -85,B 0,C 180,E1 -4387.021,E2 -4387.021} C_VEL
LIN {X 0,Y 530.973,Z 320.961,A -85,B 0,C 180,E1 -4389.467,E2 -4389.467} C_VEL
LIN {X 0,Y 530.883,Z 325.392,A -85,B 0,C 180,E1 -4390.906,E2 -4390.906} C_VEL
LIN {X 0,Y 534.22,Z 340.146,A -85,B 0,C 180,E1 -4391.299,E2 -4391.299} C_VEL
LIN {X 0,Y 533.892,Z 355.9,A -85,B 0,C 180,E1 -4391.719,E2 -4391.719} C_VEL
LIN {X 0,Y 533.546,Z 370.934,A -85,B 0,C 180,E1 -4392.287,E2 -4392.287} C_VEL
LIN {X 0,Y 533.148,Z 384.379,A -85,B 0,C 180,E1 -4392.945,E2 -4392.945} C_VEL
LIN {X 0,Y 532.689,Z 398.636,A -85,B 0,C 180,E1 -4393.817,E2 -4393.817} C_VEL
LIN {X 0,Y 532.288,Z 411.539,A -85,B 0,C 180,E1 -4394.787,E2 -4394.787} C_VEL
LIN {X 0,Y 531.831,Z 423.339,A -85,B 0,C 180,E1 -4395.85,E2 -4395.85} C_VEL
LIN {X 0,Y 531.493,Z 434.143,A -85,B 0,C 180,E1 -4397.01,E2 -4397.01} C_VEL
LIN {X 0,Y 531.107,Z 444.259,A -85,B 0,C 180,E1 -4398.3,E2 -4398.3} C_VEL
LIN {X 0,Y 530.941,Z 453.419,A -85,B 0,C 180,E1 -4399.707,E2 -4399.707} C_VEL
LIN {X 0,Y 530.759,Z 459.754,A -85,B 0,C 180,E1 -4400.858,E2 -4400.858} C_VEL
LIN {X 0,Y 530.601,Z 466.704,A -85,B 0,C 180,E1 -4402.389,E2 -4402.389} C_VEL
LIN {X 0,Y 530.529,Z 472.164,A -85,B 0,C 180,E1 -4403.917,E2 -4403.917} C_VEL
LIN {X 0,Y 530.413,Z 476.293,A -85,B 0,C 180,E1 -4405.441,E2 -4405.441} C_VEL
LIN {X 0,Y 530.448,Z 479.188,A -85,B 0,C 180,E1 -4406.963,E2 -4406.963} C_VEL
LIN {X 0,Y 530.358,Z 480.911,A -85,B 0,C 180,E1 -4408.482,E2 -4408.482} C_VEL
LIN {X 0,Y 530.34,Z 481.5,A -85,B 0,C 180,E1 -4410.001,E2 -4410.001} C_VEL
LIN {X 0,Y 530.358,Z 480.909,A -85,B 0,C 180,E1 -4411.519,E2 -4411.519} C_VEL
LIN {X 0,Y 530.449,Z 479.184,A -85,B 0,C 180,E1 -4413.038,E2 -4413.038} C_VEL
LIN {X 0,Y 530.413,Z 476.288,A -85,B 0,C 180,E1 -4414.56,E2 -4414.56} C_VEL
LIN {X 0,Y 530.522,Z 472.162,A -85,B 0,C 180,E1 -4416.084,E2 -4416.084} C_VEL
LIN {X 0,Y 530.602,Z 466.7,A -85,B 0,C 180,E1 -4417.612,E2 -4417.612} C_VEL
LIN {X 0,Y 530.76,Z 459.745,A -85,B 0,C 180,E1 -4419.143,E2 -4419.143} C_VEL
LIN {X 0,Y 530.98,Z 452.289,A -85,B 0,C 180,E1 -4420.486,E2 -4420.486} C_VEL
LIN {X 0,Y 531.174,Z 442.953,A -85,B 0,C 180,E1 -4421.884,E2 -4421.884} C_VEL
LIN {X 0,Y 531.565,Z 432.504,A -85,B 0,C 180,E1 -4423.184,E2 -4423.184} C_VEL
LIN {X 0,Y 531.905,Z 421.38,A -85,B 0,C 180,E1 -4424.344,E2 -4424.344} C_VEL
LIN {X 0,Y 532.36,Z 409.259,A -85,B 0,C 180,E1 -4425.402,E2 -4425.402} C_VEL
LIN {X 0,Y 532.772,Z 395.769,A -85,B 0,C 180,E1 -4426.378,E2 -4426.378} C_VEL
LIN {X 0,Y 533.194,Z 382.589,A -85,B 0,C 180,E1 -4427.153,E2 -4427.153} C_VEL
LIN {X 0,Y 533.607,Z 369.163,A -85,B 0,C 180,E1 -4427.788,E2 -4427.788} C_VEL
LIN {X 0,Y 533.952,Z 354.351,A -85,B 0,C 180,E1 -4428.329,E2 -4428.329} C_VEL
LIN {X 0,Y 534.134,Z 338.984,A -85,B 0,C 180,E1 -4428.729,E2 -4428.729} C_VEL
LIN {X 0,Y 530.893,Z 325.38,A -85,B 0,C 180,E1 -4429.097,E2 -4429.097} C_VEL
LIN {X 0,Y 531.026,Z 316.145,A -85,B 0,C 180,E1 -4432.114,E2 -4432.114} C_VEL
LIN {X 0,Y 531.189,Z 307.341,A -85,B 0,C 180,E1 -4435.049,E2 -4435.049} C_VEL
LIN {X 0,Y 531.419,Z 298.678,A -85,B 0,C 180,E1 -4438.001,E2 -4438.001} C_VEL
LIN {X 0,Y 531.562,Z 290.823,A -85,B 0,C 180,E1 -4440.751,E2 -4440.751} C_VEL
LIN {X 0,Y 531.799,Z 282.488,A -85,B 0,C 180,E1 -4443.715,E2 -4443.715} C_VEL
LIN {X 0,Y 531.995,Z 273.6,A -85,B 0,C 180,E1 -4446.948,E2 -4446.948} C_VEL
LIN {X 0,Y 532.161,Z 267.234,A -85,B 0,C 180,E1 -4449.34,E2 -4449.34} C_VEL
LIN {X 0,Y 532.165,Z 260.934,A -85,B 0,C 180,E1 -4451.797,E2 -4451.797} C_VEL
LIN {X 0,Y 531.402,Z 256.122,A -85,B 0,C 180,E1 -4453.919,E2 -4453.919} C_VEL
LIN {X 0,Y 530.986,Z 253.971,A -85,B 0,C 180,E1 -4454.985,E2 -4454.985} C_VEL
LIN {X 0,Y 530.986,Z 253.97,A -85,B 0,C 180,E1 -4457.834,E2 -4457.834} C_VEL
LIN {X 0,Y 530.991,Z 253.971,A -85,B 0,C 180,E1 -4460.557,E2 -4460.557} C_VEL
LIN {X 0,Y 530.96,Z 253.974,A -85,B 0,C 180,E1 -4463.441,E2 -4463.441} C_VEL
LIN {X 0,Y 530.961,Z 253.972,A -85,B 0,C 180,E1 -4466.225,E2 -4466.225} C_VEL
LIN {X 0,Y 530.98,Z 253.97,A -85,B 0,C 180,E1 -4469.355,E2 -4469.355} C_VEL
LIN {X 0,Y 531.019,Z 253.966,A -85,B 0,C 180,E1 -4472.467,E2 -4472.467} C_VEL
LIN {X 0,Y 531.011,Z 253.968,A -85,B 0,C 180,E1 -4474.942,E2 -4474.942} C_VEL
LIN {X 0,Y 530.977,Z 253.972,A -85,B 0,C 180,E1 -4478.246,E2 -4478.246} C_VEL
LIN {X 0,Y 531.001,Z 253.969,A -85,B 0,C 180,E1 -4480.677,E2 -4480.677} C_VEL
LIN {X 0,Y 530.991,Z 253.97,A -85,B 0,C 180,E1 -4483.071,E2 -4483.071} C_VEL
LIN {X 0,Y 531.024,Z 253.966,A -85,B 0,C 180,E1 -4485.435,E2 -4485.435} C_VEL
LIN {X 0,Y 531.042,Z 253.964,A -85,B 0,C 180,E1 -4488.549,E2 -4488.549} C_VEL
LIN {X 0,Y 531.058,Z 253.961,A -85,B 0,C 180,E1 -4491.629,E2 -4491.629} C_VEL
LIN {X 0,Y 531.121,Z 253.954,A -85,B 0,C 180,E1 -4494.685,E2 -4494.685} C_VEL
LIN {X 0,Y 531.143,Z 253.949,A -85,B 0,C 180,E1 -4497.724,E2 -4497.724} C_VEL
LIN {X 0,Y 531.158,Z 253.949,A -85,B 0,C 180,E1 -4500.757,E2 -4500.757} C_VEL
LIN {X 0,Y 531.108,Z 253.955,A -85,B 0,C 180,E1 -4503.033,E2 -4503.033} C_VEL
LIN {X 0,Y 531.085,Z 253.958,A -85,B 0,C 180,E1 -4506.076,E2 -4506.076} C_VEL
LIN {X 0,Y 531.031,Z 253.963,A -85,B 0,C 180,E1 -4509.137,E2 -4509.137} C_VEL
LIN {X 0,Y 531.043,Z 253.963,A -85,B 0,C 180,E1 -4512.224,E2 -4512.224} C_VEL
LIN {X 0,Y 530.998,Z 253.967,A -85,B 0,C 180,E1 -4515.349,E2 -4515.349} C_VEL
LIN {X 0,Y 530.992,Z 253.969,A -85,B 0,C 180,E1 -4518.52,E2 -4518.52} C_VEL
LIN {X 0,Y 530.999,Z 253.969,A -85,B 0,C 180,E1 -4520.937,E2 -4520.937} C_VEL
LIN {X 0,Y 530.98,Z 253.973,A -85,B 0,C 180,E1 -4524.223,E2 -4524.223} C_VEL
LIN {X 0,Y 531.006,Z 253.967,A -85,B 0,C 180,E1 -4526.742,E2 -4526.742} C_VEL
LIN {X 0,Y 530.981,Z 253.97,A -85,B 0,C 180,E1 -4529.321,E2 -4529.321} C_VEL
LIN {X 0,Y 530.969,Z 253.972,A -85,B 0,C 180,E1 -4532.1,E2 -4532.1} C_VEL
LIN {X 0,Y 530.987,Z 253.97,A -85,B 0,C 180,E1 -4534.853,E2 -4534.853} C_VEL
LIN {X 0,Y 530.964,Z 253.973,A -85,B 0,C 180,E1 -4537.506,E2 -4537.506} C_VEL
LIN {X 0,Y 530.981,Z 253.97,A -85,B 0,C 180,E1 -4540.431,E2 -4540.431} C_VEL
LIN {X 0,Y 530.966,Z 253.973,A -85,B 0,C 180,E1 -4543.281,E2 -4543.281} C_VEL
LIN {X 0,Y 530.959,Z 253.973,A -85,B 0,C 180,E1 -4543.563,E2 -4543.563} C_VEL
LIN {X 0,Y 530.286,Z 254.058,A -85,B 0,C 180,E1 -4544.196,E2 -4544.196} C_VEL
LIN {X 0,Y 527.439,Z 254.413,A -85,B 0,C 180,E1 -4545.225,E2 -4545.225} C_VEL
LIN {X 0,Y 525.037,Z 254.713,A -85,B 0,C 180,E1 -4546.054,E2 -4546.054} C_VEL
LIN {X 0,Y 524.004,Z 254.839,A -85,B 0,C 180,E1 -4546.693,E2 -4546.693} C_VEL
LIN {X 0,Y 523.918,Z 254.849,A -85,B 0,C 180,E1 -4546.91,E2 -4546.91} C_VEL
LIN {X 0,Y 523.973,Z 254.844,A -85,B 0,C 180,E1 -4549.922,E2 -4549.922} C_VEL
LIN {X 0,Y 523.906,Z 254.851,A -85,B 0,C 180,E1 -4552.867,E2 -4552.867} C_VEL
LIN {X 0,Y 523.937,Z 254.85,A -85,B 0,C 180,E1 -4555.71,E2 -4555.71} C_VEL
LIN {X 0,Y 523.926,Z 254.85,A -85,B 0,C 180,E1 -4558.456,E2 -4558.456} C_VEL
LIN {X 0,Y 523.944,Z 254.848,A -85,B 0,C 180,E1 -4561.125,E2 -4561.125} C_VEL
LIN {X 0,Y 523.977,Z 254.844,A -85,B 0,C 180,E1 -4563.979,E2 -4563.979} C_VEL
LIN {X 0,Y 523.928,Z 254.848,A -85,B 0,C 180,E1 -4566.27,E2 -4566.27} C_VEL
LIN {X 0,Y 523.938,Z 254.847,A -85,B 0,C 180,E1 -4568.766,E2 -4568.766} C_VEL
LIN {X 0,Y 523.945,Z 254.848,A -85,B 0,C 180,E1 -4571.22,E2 -4571.22} C_VEL
LIN {X 0,Y 523.931,Z 254.849,A -85,B 0,C 180,E1 -4573.638,E2 -4573.638} C_VEL
LIN {X 0,Y 523.937,Z 254.848,A -85,B 0,C 180,E1 -4576.027,E2 -4576.027} C_VEL
LIN {X 0,Y 524.001,Z 254.84,A -85,B 0,C 180,E1 -4578.393,E2 -4578.393} C_VEL
LIN {X 0,Y 523.999,Z 254.841,A -85,B 0,C 180,E1 -4581.515,E2 -4581.515} C_VEL
LIN {X 0,Y 524.037,Z 254.836,A -85,B 0,C 180,E1 -4583.84,E2 -4583.84} C_VEL
LIN {X 0,Y 523.755,Z 254.873,A -85,B 0,C 180,E1 -4586.152,E2 -4586.152} C_VEL
LIN {X 0,Y 523.658,Z 255.181,A -85,B 0,C 180,E1 -4587.692,E2 -4587.692} C_VEL
LIN {X 0,Y 523.85,Z 257.386,A -85,B 0,C 180,E1 -4589.999,E2 -4589.999} C_VEL
LIN {X 0,Y 523.602,Z 261.118,A -85,B 0,C 180,E1 -4593.848,E2 -4593.848} C_VEL
LIN {X 0,Y 523.541,Z 264.112,A -85,B 0,C 180,E1 -4596.939,E2 -4596.939} C_VEL
LIN {X 0,Y 523.46,Z 267.111,A -85,B 0,C 180,E1 -4600.051,E2 -4600.051} C_VEL
LIN {X 0,Y 523.451,Z 269.391,A -85,B 0,C 180,E1 -4602.404,E2 -4602.404} C_VEL
LIN {X 0,Y 523.41,Z 270.692,A -85,B 0,C 180,E1 -4603.738,E2 -4603.738} C_VEL
LIN {X 0,Y 527.256,Z 284.925,A -85,B 0,C 180,E1 -4604.177,E2 -4604.177} C_VEL
LIN {X 0,Y 527.314,Z 291.051,A -85,B 0,C 180,E1 -4604.348,E2 -4604.348} C_VEL
LIN {X 0,Y 526.954,Z 305.262,A -85,B 0,C 180,E1 -4604.827,E2 -4604.827} C_VEL
LIN {X 0,Y 526.515,Z 319.911,A -85,B 0,C 180,E1 -4605.483,E2 -4605.483} C_VEL
LIN {X 0,Y 526.043,Z 334.066,A -85,B 0,C 180,E1 -4606.293,E2 -4606.293} C_VEL
LIN {X 0,Y 525.636,Z 346.957,A -85,B 0,C 180,E1 -4607.206,E2 -4607.206} C_VEL
LIN {X 0,Y 525.195,Z 358.436,A -85,B 0,C 180,E1 -4608.181,E2 -4608.181} C_VEL
LIN {X 0,Y 524.73,Z 370.054,A -85,B 0,C 180,E1 -4609.359,E2 -4609.359} C_VEL
LIN {X 0,Y 524.322,Z 380.311,A -85,B 0,C 180,E1 -4610.6,E2 -4610.6} C_VEL
LIN {X 0,Y 524.016,Z 389.011,A -85,B 0,C 180,E1 -4611.849,E2 -4611.849} C_VEL
LIN {X 0,Y 523.75,Z 397.521,A -85,B 0,C 180,E1 -4613.318,E2 -4613.318} C_VEL
LIN {X 0,Y 523.583,Z 403.644,A -85,B 0,C 180,E1 -4614.589,E2 -4614.589} C_VEL
LIN {X 0,Y 523.481,Z 410.299,A -85,B 0,C 180,E1 -4616.297,E2 -4616.297} C_VEL
LIN {X 0,Y 523.388,Z 414.241,A -85,B 0,C 180,E1 -4617.599,E2 -4617.599} C_VEL
LIN {X 0,Y 523.305,Z 417.891,A -85,B 0,C 180,E1 -4619.2,E2 -4619.2} C_VEL
LIN {X 0,Y 523.264,Z 420.181,A -85,B 0,C 180,E1 -4620.732,E2 -4620.732} C_VEL
LIN {X 0,Y 523.249,Z 421.392,A -85,B 0,C 180,E1 -4622.496,E2 -4622.496} C_VEL
LIN {X 0,Y 523.267,Z 421.387,A -85,B 0,C 180,E1 -4623.623,E2 -4623.623} C_VEL
LIN {X 0,Y 523.255,Z 420.268,A -85,B 0,C 180,E1 -4625.277,E2 -4625.277} C_VEL
LIN {X 0,Y 523.25,Z 418.918,A -85,B 0,C 180,E1 -4626.306,E2 -4626.306} C_VEL
LIN {X 0,Y 523.293,Z 416.462,A -85,B 0,C 180,E1 -4627.593,E2 -4627.593} C_VEL
LIN {X 0,Y 523.408,Z 412.425,A -85,B 0,C 180,E1 -4629.13,E2 -4629.13} C_VEL
LIN {X 0,Y 523.49,Z 406.234,A -85,B 0,C 180,E1 -4630.88,E2 -4630.88} C_VEL
LIN {X 0,Y 523.684,Z 399.285,A -85,B 0,C 180,E1 -4632.431,E2 -4632.431} C_VEL
LIN {X 0,Y 523.94,Z 391.348,A -85,B 0,C 180,E1 -4633.87,E2 -4633.87} C_VEL
LIN {X 0,Y 524.257,Z 381.974,A -85,B 0,C 180,E1 -4635.275,E2 -4635.275} C_VEL
LIN {X 0,Y 524.63,Z 372.342,A -85,B 0,C 180,E1 -4636.485,E2 -4636.485} C_VEL
LIN {X 0,Y 525.105,Z 360.633,A -85,B 0,C 180,E1 -4637.713,E2 -4637.713} C_VEL
LIN {X 0,Y 525.591,Z 348.265,A -85,B 0,C 180,E1 -4638.791,E2 -4638.791} C_VEL
LIN {X 0,Y 526.104,Z 335.272,A -85,B 0,C 180,E1 -4639.726,E2 -4639.726} C_VEL
LIN {X 0,Y 526.547,Z 321.471,A -85,B 0,C 180,E1 -4640.534,E2 -4640.534} C_VEL
LIN {X 0,Y 526.959,Z 307.408,A -85,B 0,C 180,E1 -4641.185,E2 -4641.185} C_VEL
LIN {X 0,Y 527.342,Z 292.418,A -85,B 0,C 180,E1 -4641.707,E2 -4641.707} C_VEL
LIN {X 0,Y 527.281,Z 284.943,A -85,B 0,C 180,E1 -4641.915,E2 -4641.915} C_VEL
LIN {X 0,Y 524.159,Z 273.576,A -85,B 0,C 180,E1 -4642.268,E2 -4642.268} C_VEL
LIN {X 0,Y 523.441,Z 270.989,A -85,B 0,C 180,E1 -4642.348,E2 -4642.348} C_VEL
LIN {X 0,Y 523.488,Z 267.91,A -85,B 0,C 180,E1 -4645.678,E2 -4645.678} C_VEL
LIN {X 0,Y 523.555,Z 265.352,A -85,B 0,C 180,E1 -4648.433,E2 -4648.433} C_VEL
LIN {X 0,Y 523.612,Z 262.889,A -85,B 0,C 180,E1 -4651.107,E2 -4651.107} C_VEL
LIN {X 0,Y 523.644,Z 260.193,A -85,B 0,C 180,E1 -4654.055,E2 -4654.055} C_VEL
LIN {X 0,Y 523.697,Z 258.131,A -85,B 0,C 180,E1 -4656.26,E2 -4656.26} C_VEL
LIN {X 0,Y 523.71,Z 255.803,A -85,B 0,C 180,E1 -4658.758,E2 -4658.758} C_VEL
LIN {X 0,Y 523.749,Z 254.874,A -85,B 0,C 180,E1 -4659.933,E2 -4659.933} C_VEL
LIN {X 0,Y 523.943,Z 254.849,A -85,B 0,C 180,E1 -4662.838,E2 -4662.838} C_VEL
LIN {X 0,Y 523.97,Z 254.845,A -85,B 0,C 180,E1 -4665.237,E2 -4665.237} C_VEL
LIN {X 0,Y 524.006,Z 254.84,A -85,B 0,C 180,E1 -4668.395,E2 -4668.395} C_VEL
LIN {X 0,Y 524,Z 254.84,A -85,B 0,C 180,E1 -4671.517,E2 -4671.517} C_VEL
LIN {X 0,Y 524.08,Z 254.83,A -85,B 0,C 180,E1 -4674.615,E2 -4674.615} C_VEL
LIN {X 0,Y 524.109,Z 254.826,A -85,B 0,C 180,E1 -4677.695,E2 -4677.695} C_VEL
LIN {X 0,Y 524.12,Z 254.825,A -85,B 0,C 180,E1 -4680.769,E2 -4680.769} C_VEL
LIN {X 0,Y 524.07,Z 254.831,A -85,B 0,C 180,E1 -4683.076,E2 -4683.076} C_VEL
LIN {X 0,Y 524.043,Z 254.834,A -85,B 0,C 180,E1 -4686.16,E2 -4686.16} C_VEL
LIN {X 0,Y 523.999,Z 254.84,A -85,B 0,C 180,E1 -4689.263,E2 -4689.263} C_VEL
LIN {X 0,Y 524,Z 254.84,A -85,B 0,C 180,E1 -4691.741,E2 -4691.741} C_VEL
LIN {X 0,Y 523.99,Z 254.842,A -85,B 0,C 180,E1 -4695.053,E2 -4695.053} C_VEL
LIN {X 0,Y 523.961,Z 254.844,A -85,B 0,C 180,E1 -4697.97,E2 -4697.97} C_VEL
LIN {X 0,Y 523.97,Z 254.846,A -85,B 0,C 180,E1 -4700.411,E2 -4700.411} C_VEL
LIN {X 0,Y 523.915,Z 254.851,A -85,B 0,C 180,E1 -4702.894,E2 -4702.894} C_VEL
LIN {X 0,Y 523.953,Z 254.846,A -85,B 0,C 180,E1 -4705.419,E2 -4705.419} C_VEL
LIN {X 0,Y 523.968,Z 254.846,A -85,B 0,C 180,E1 -4708,E2 -4708} C_VEL
LIN {X 0,Y 523.942,Z 254.85,A -85,B 0,C 180,E1 -4710.855,E2 -4710.855} C_VEL
LIN {X 0,Y 523.957,Z 254.848,A -85,B 0,C 180,E1 -4713.735,E2 -4713.735} C_VEL
LIN {X 0,Y 523.901,Z 254.856,A -85,B 0,C 180,E1 -4716.402,E2 -4716.402} C_VEL
LIN {X 0,Y 523.922,Z 254.853,A -85,B 0,C 180,E1 -4719.085,E2 -4719.085} C_VEL
LIN {X 0,Y 523.951,Z 254.847,A -85,B 0,C 180,E1 -4722.119,E2 -4722.119} C_VEL
LIN {X 0,Y 523.984,Z 254.996,A -85,B 0,C 180,E1 -4724.964,E2 -4724.964} C_VEL
LIN {X 0,Y 524.937,Z 260.404,A -85,B 0,C 180,E1 -4727.422,E2 -4727.422} C_VEL
LIN {X 0,Y 525.231,Z 264.226,A -85,B 0,C 180,E1 -4729.031,E2 -4729.031} C_VEL
LIN {X 0,Y 525.067,Z 270.413,A -85,B 0,C 180,E1 -4731.509,E2 -4731.509} C_VEL
LIN {X 0,Y 524.841,Z 278.142,A -85,B 0,C 180,E1 -4734.375,E2 -4734.375} C_VEL
LIN {X 0,Y 524.702,Z 285.992,A -85,B 0,C 180,E1 -4737.149,E2 -4737.149} C_VEL
LIN {X 0,Y 524.513,Z 294.967,A -85,B 0,C 180,E1 -4740.28,E2 -4740.28} C_VEL
LIN {X 0,Y 524.322,Z 302.394,A -85,B 0,C 180,E1 -4742.888,E2 -4742.888} C_VEL
LIN {X 0,Y 524.132,Z 310.75,A -85,B 0,C 180,E1 -4745.756,E2 -4745.756} C_VEL
LIN {X 0,Y 523.983,Z 319.723,A -85,B 0,C 180,E1 -4748.769,E2 -4748.769} C_VEL
LIN {X 0,Y 523.869,Z 325.411,A -85,B 0,C 180,E1 -4750.647,E2 -4750.647} C_VEL
LIN {X 0,Y 527.505,Z 340.51,A -85,B 0,C 180,E1 -4751.06,E2 -4751.06} C_VEL
LIN {X 0,Y 527.171,Z 355.899,A -85,B 0,C 180,E1 -4751.478,E2 -4751.478} C_VEL
LIN {X 0,Y 526.78,Z 371.011,A -85,B 0,C 180,E1 -4752.056,E2 -4752.056} C_VEL
LIN {X 0,Y 526.35,Z 384.378,A -85,B 0,C 180,E1 -4752.718,E2 -4752.718} C_VEL
LIN {X 0,Y 525.92,Z 397.21,A -85,B 0,C 180,E1 -4753.503,E2 -4753.503} C_VEL
LIN {X 0,Y 525.422,Z 410.364,A -85,B 0,C 180,E1 -4754.484,E2 -4754.484} C_VEL
LIN {X 0,Y 524.979,Z 421.387,A -85,B 0,C 180,E1 -4755.463,E2 -4755.463} C_VEL
LIN {X 0,Y 524.598,Z 432.514,A -85,B 0,C 180,E1 -4756.639,E2 -4756.639} C_VEL
LIN {X 0,Y 524.154,Z 443.311,A -85,B 0,C 180,E1 -4758.006,E2 -4758.006} C_VEL
LIN {X 0,Y 523.943,Z 452.298,A -85,B 0,C 180,E1 -4759.372,E2 -4759.372} C_VEL
LIN {X 0,Y 523.699,Z 459.753,A -85,B 0,C 180,E1 -4760.733,E2 -4760.733} C_VEL
LIN {X 0,Y 523.535,Z 466.704,A -85,B 0,C 180,E1 -4762.286,E2 -4762.286} C_VEL
LIN {X 0,Y 523.441,Z 472.164,A -85,B 0,C 180,E1 -4763.834,E2 -4763.834} C_VEL
LIN {X 0,Y 523.323,Z 476.293,A -85,B 0,C 180,E1 -4765.379,E2 -4765.379} C_VEL
LIN {X 0,Y 523.358,Z 479.187,A -85,B 0,C 180,E1 -4766.921,E2 -4766.921} C_VEL
LIN {X 0,Y 523.272,Z 480.911,A -85,B 0,C 180,E1 -4768.461,E2 -4768.461} C_VEL
LIN {X 0,Y 523.243,Z 481.5,A -85,B 0,C 180,E1 -4770.001,E2 -4770.001} C_VEL
LIN {X 0,Y 523.272,Z 480.909,A -85,B 0,C 180,E1 -4771.54,E2 -4771.54} C_VEL
LIN {X 0,Y 523.358,Z 479.183,A -85,B 0,C 180,E1 -4773.08,E2 -4773.08} C_VEL
LIN {X 0,Y 523.324,Z 476.288,A -85,B 0,C 180,E1 -4774.622,E2 -4774.622} C_VEL
LIN {X 0,Y 523.432,Z 472.162,A -85,B 0,C 180,E1 -4776.167,E2 -4776.167} C_VEL
LIN {X 0,Y 523.536,Z 466.699,A -85,B 0,C 180,E1 -4777.715,E2 -4777.715} C_VEL
LIN {X 0,Y 523.7,Z 459.744,A -85,B 0,C 180,E1 -4779.268,E2 -4779.268} C_VEL
LIN {X 0,Y 523.988,Z 451.083,A -85,B 0,C 180,E1 -4780.823,E2 -4780.823} C_VEL
LIN {X 0,Y 524.234,Z 441.845,A -85,B 0,C 180,E1 -4782.194,E2 -4782.194} C_VEL
LIN {X 0,Y 524.6,Z 432.504,A -85,B 0,C 180,E1 -4783.362,E2 -4783.362} C_VEL
LIN {X 0,Y 525.014,Z 420.349,A -85,B 0,C 180,E1 -4784.636,E2 -4784.636} C_VEL
LIN {X 0,Y 525.485,Z 408.824,A -85,B 0,C 180,E1 -4785.645,E2 -4785.645} C_VEL
LIN {X 0,Y 525.906,Z 395.768,A -85,B 0,C 180,E1 -4786.598,E2 -4786.598} C_VEL
LIN {X 0,Y 526.375,Z 382.588,A -85,B 0,C 180,E1 -4787.383,E2 -4787.383} C_VEL
LIN {X 0,Y 526.839,Z 369.3,A -85,B 0,C 180,E1 -4788.018,E2 -4788.018} C_VEL
LIN {X 0,Y 527.218,Z 354.528,A -85,B 0,C 180,E1 -4788.566,E2 -4788.566} C_VEL
LIN {X 0,Y 527.375,Z 340.005,A -85,B 0,C 180,E1 -4788.956,E2 -4788.956} C_VEL
LIN {X 0,Y 523.852,Z 325.428,A -85,B 0,C 180,E1 -4789.348,E2 -4789.348} C_VEL
LIN {X 0,Y 523.985,Z 316.642,A -85,B 0,C 180,E1 -4792.261,E2 -4792.261} C_VEL
LIN {X 0,Y 524.207,Z 307.341,A -85,B 0,C 180,E1 -4795.406,E2 -4795.406} C_VEL
LIN {X 0,Y 524.441,Z 298.677,A -85,B 0,C 180,E1 -4798.408,E2 -4798.408} C_VEL
LIN {X 0,Y 524.617,Z 289.924,A -85,B 0,C 180,E1 -4801.498,E2 -4801.498} C_VEL
LIN {X 0,Y 524.811,Z 282.325,A -85,B 0,C 180,E1 -4804.225,E2 -4804.225} C_VEL
LIN {X 0,Y 525.114,Z 273.682,A -85,B 0,C 180,E1 -4807.441,E2 -4807.441} C_VEL
LIN {X 0,Y 525.264,Z 266.249,A -85,B 0,C 180,E1 -4810.301,E2 -4810.301} C_VEL
LIN {X 0,Y 525.193,Z 262.028,A -85,B 0,C 180,E1 -4811.997,E2 -4811.997} C_VEL
LIN {X 0,Y 524.14,Z 255.961,A -85,B 0,C 180,E1 -4814.711,E2 -4814.711} C_VEL
LIN {X 0,Y 523.959,Z 254.847,A -85,B 0,C 180,E1 -4815.309,E2 -4815.309} C_VEL
LIN {X 0,Y 523.96,Z 254.846,A -85,B 0,C 180,E1 -4818.69,E2 -4818.69} C_VEL
LIN {X 0,Y 523.922,Z 254.85,A -85,B 0,C 180,E1 -4821.081,E2 -4821.081} C_VEL
LIN {X 0,Y 523.905,Z 254.852,A -85,B 0,C 180,E1 -4823.825,E2 -4823.825} C_VEL
LIN {X 0,Y 523.918,Z 254.851,A -85,B 0,C 180,E1 -4826.633,E2 -4826.633} C_VEL
LIN {X 0,Y 523.961,Z 254.845,A -85,B 0,C 180,E1 -4829.356,E2 -4829.356} C_VEL
LIN {X 0,Y 523.981,Z 254.843,A -85,B 0,C 180,E1 -4832.281,E2 -4832.281} C_VEL
LIN {X 0,Y 523.958,Z 254.846,A -85,B 0,C 180,E1 -4834.581,E2 -4834.581} C_VEL
LIN {X 0,Y 523.917,Z 254.852,A -85,B 0,C 180,E1 -4837.106,E2 -4837.106} C_VEL
LIN {X 0,Y 523.985,Z 254.841,A -85,B 0,C 180,E1 -4839.866,E2 -4839.866} C_VEL
LIN {X 0,Y 523.973,Z 254.844,A -85,B 0,C 180,E1 -4842.837,E2 -4842.837} C_VEL
LIN {X 0,Y 523.982,Z 254.843,A -85,B 0,C 180,E1 -4845.235,E2 -4845.235} C_VEL
LIN {X 0,Y 524.018,Z 254.838,A -85,B 0,C 180,E1 -4848.394,E2 -4848.394} C_VEL
LIN {X 0,Y 524.006,Z 254.839,A -85,B 0,C 180,E1 -4851.515,E2 -4851.515} C_VEL
LIN {X 0,Y 524.081,Z 254.831,A -85,B 0,C 180,E1 -4854.613,E2 -4854.613} C_VEL
LIN {X 0,Y 524.116,Z 254.824,A -85,B 0,C 180,E1 -4857.694,E2 -4857.694} C_VEL
LIN {X 0,Y 524.128,Z 254.824,A -85,B 0,C 180,E1 -4860.767,E2 -4860.767} C_VEL
LIN {X 0,Y 524.074,Z 254.832,A -85,B 0,C 180,E1 -4863.074,E2 -4863.074} C_VEL
LIN {X 0,Y 524.048,Z 254.835,A -85,B 0,C 180,E1 -4866.158,E2 -4866.158} C_VEL
LIN {X 0,Y 524.005,Z 254.842,A -85,B 0,C 180,E1 -4868.483,E2 -4868.483} C_VEL
LIN {X 0,Y 524.006,Z 254.84,A -85,B 0,C 180,E1 -4871.738,E2 -4871.738} C_VEL
LIN {X 0,Y 523.995,Z 254.84,A -85,B 0,C 180,E1 -4875.051,E2 -4875.051} C_VEL
LIN {X 0,Y 523.966,Z 254.846,A -85,B 0,C 180,E1 -4877.968,E2 -4877.968} C_VEL
LIN {X 0,Y 523.972,Z 254.844,A -85,B 0,C 180,E1 -4880.409,E2 -4880.409} C_VEL
LIN {X 0,Y 523.917,Z 254.851,A -85,B 0,C 180,E1 -4882.892,E2 -4882.892} C_VEL
LIN {X 0,Y 523.953,Z 254.847,A -85,B 0,C 180,E1 -4885.417,E2 -4885.417} C_VEL
